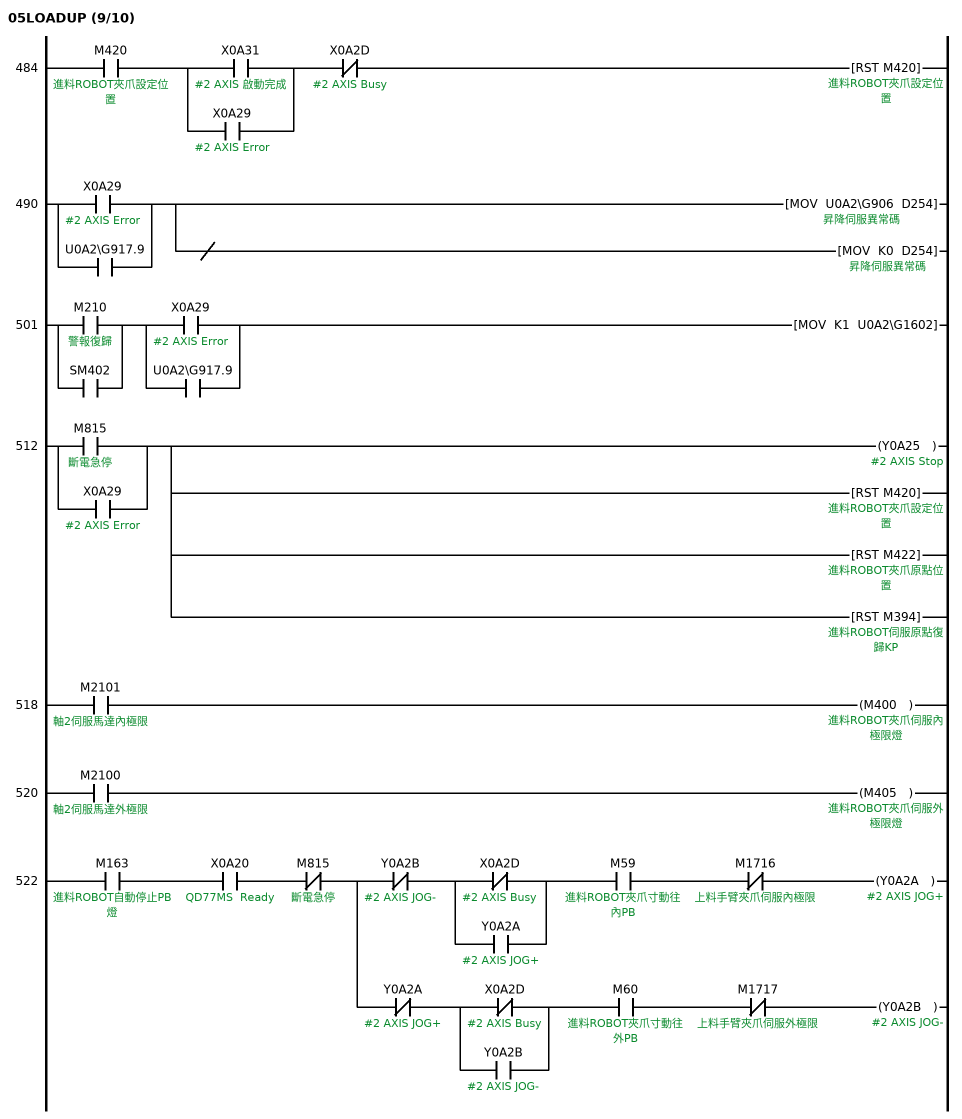
[picture p24: ladder of 05LOADUP, rungs at steps 484 to 522]
484   LD      M420  ; 進料ROBOT夾爪設定位置
      LD      X0A31  ; #2 AXIS 啟動完成
      OR      X0A29  ; #2 AXIS Error
      ANB
      ANI     X0A2D  ; #2 AXIS Busy
      RST     M420  ; 進料ROBOT夾爪設定位置
490   LD      X0A29  ; #2 AXIS Error
      OR      U0A2\G917.9
      MOV     U0A2\G906 D254  ; 昇降伺服異常碼
      INV
      MOV     K0 D254
501   LD      M210  ; 警報復歸
      OR      SM402
      LD      X0A29  ; #2 AXIS Error
      OR      U0A2\G917.9
      ANB
      MOV     K1 U0A2\G1602
512   LD      M815  ; 斷電急停
      OR      X0A29  ; #2 AXIS Error
      OUT     Y0A25  ; #2 AXIS Stop
      RST     M420  ; 進料ROBOT夾爪設定位置
      RST     M422  ; 進料ROBOT夾爪原點位置
      RST     M394  ; 進料ROBOT伺服原點復歸KP
518   LD      M2101  ; 軸2伺服馬達內極限
      OUT     M400  ; 進料ROBOT夾爪伺服內極限燈
520   LD      M2100  ; 軸2伺服馬達外極限
      OUT     M405  ; 進料ROBOT夾爪伺服外極限燈
522   LD      M163  ; 進料ROBOT自動停止PB燈
      AND     X0A20  ; QD77MS  Ready
      ANI     M815  ; 斷電急停
      MPS
      ANI     Y0A2B  ; #2 AXIS JOG-
      LDI     X0A2D  ; #2 AXIS Busy
      OR      Y0A2A  ; #2 AXIS JOG+
      ANB
      AND     M59  ; 進料ROBOT夾爪寸動往內PB
      ANI     M1716  ; 上料手臂夾爪伺服內極限
      OUT     Y0A2A  ; #2 AXIS JOG+
      MPP
      ANI     Y0A2A  ; #2 AXIS JOG+
      LDI     X0A2D  ; #2 AXIS Busy
      OR      Y0A2B  ; #2 AXIS JOG-
      ANB
      AND     M60  ; 進料ROBOT夾爪寸動往外PB
      ANI     M1717  ; 上料手臂夾爪伺服外極限
      OUT     Y0A2B  ; #2 AXIS JOG-
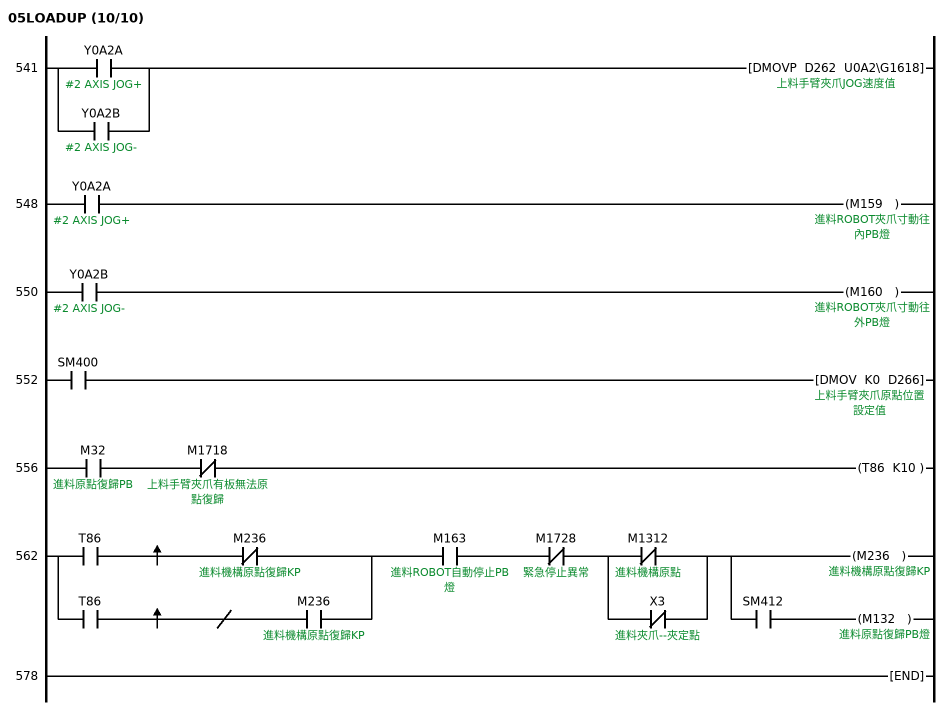
541   LD      Y0A2A  ; #2 AXIS JOG+
      OR      Y0A2B  ; #2 AXIS JOG-
      DMOVP   D262 U0A2\G1618  ; 上料手臂夾爪JOG速度值
548   LD      Y0A2A  ; #2 AXIS JOG+
      OUT     M159  ; 進料ROBOT夾爪寸動往內PB燈
550   LD      Y0A2B  ; #2 AXIS JOG-
      OUT     M160  ; 進料ROBOT夾爪寸動往外PB燈
552   LD      SM400
      DMOV    K0 D266
556   LD      M32  ; 進料原點復歸PB
      ANI     M1718  ; 上料手臂夾爪有板無法原點復歸
      OUT     T86 K10
562   LD      T86
      MEP
      ANI     M236  ; 進料機構原點復歸KP
      LD      T86
      MEP
      INV
      AND     M236  ; 進料機構原點復歸KP
      ORB
      AND     M163  ; 進料ROBOT自動停止PB燈
      ANI     M1728  ; 緊急停止異常
      LDI     M1312  ; 進料機構原點
      ORI     X3  ; 進料夾爪--夾定點
      ANB
      OUT     M236  ; 進料機構原點復歸KP
      AND     SM412
      OUT     M132  ; 進料原點復歸PB燈
578   END
END_PROGRAM

PROGRAM 06UNLOAD
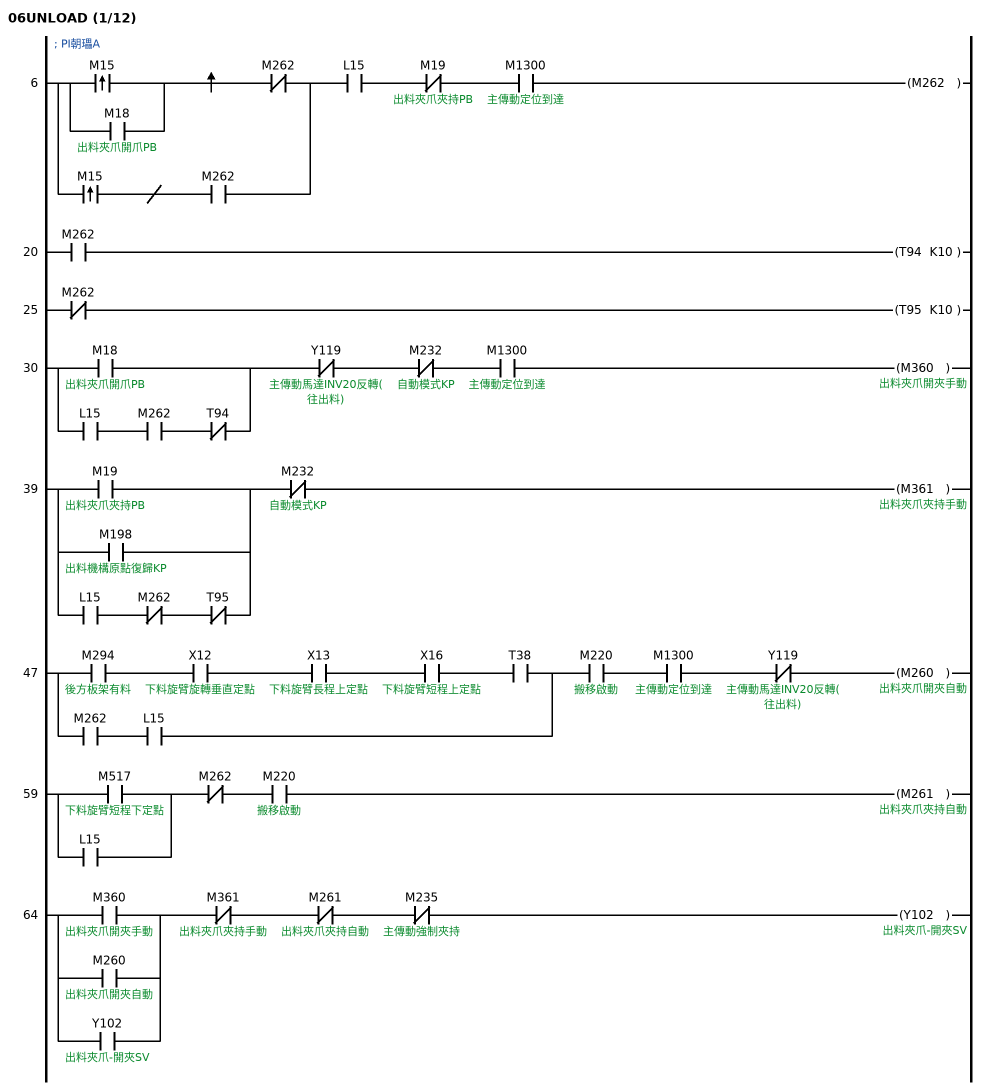
; PI朝瓃Α
6     LDP     M15
      OR      M18  ; 出料夾爪開爪PB
      MEP
      ANI     M262
      LDP     M15
      INV
      AND     M262
      ORB
      AND     L15
      ANI     M19  ; 出料夾爪夾持PB
      AND     M1300  ; 主傳動定位到達
      OUT     M262
20    LD      M262
      OUT     T94 K10
25    LDI     M262
      OUT     T95 K10
30    LD      M18  ; 出料夾爪開爪PB
      LD      L15
      AND     M262
      ANI     T94
      ORB
      ANI     Y119  ; 主傳動馬達INV20反轉(往出料)
      ANI     M232  ; 自動模式KP
      AND     M1300  ; 主傳動定位到達
      OUT     M360  ; 出料夾爪開夾手動
39    LD      M19  ; 出料夾爪夾持PB
      OR      M198  ; 出料機構原點復歸KP
      LD      L15
      ANI     M262
      ANI     T95
      ORB
      ANI     M232  ; 自動模式KP
      OUT     M361  ; 出料夾爪夾持手動
47    LD      M294  ; 後方板架有料
      AND     X12  ; 下料旋臂旋轉垂直定點
      AND     X13  ; 下料旋臂長程上定點
      AND     X16  ; 下料旋臂短程上定點
      AND     T38
      LD      M262
      AND     L15
      ORB
      AND     M220  ; 搬移啟動
      AND     M1300  ; 主傳動定位到達
      ANI     Y119  ; 主傳動馬達INV20反轉(往出料)
      OUT     M260  ; 出料夾爪開夾自動
59    LD      M517  ; 下料旋臂短程下定點
      OR      L15
      ANI     M262
      AND     M220  ; 搬移啟動
      OUT     M261  ; 出料夾爪夾持自動
64    LD      M360  ; 出料夾爪開夾手動
      OR      M260  ; 出料夾爪開夾自動
      OR      Y102  ; 出料夾爪-開夾SV
      ANI     M361  ; 出料夾爪夾持手動
      ANI     M261  ; 出料夾爪夾持自動
      ANI     M235  ; 主傳動強制夾持
      OUT     Y102  ; 出料夾爪-開夾SV
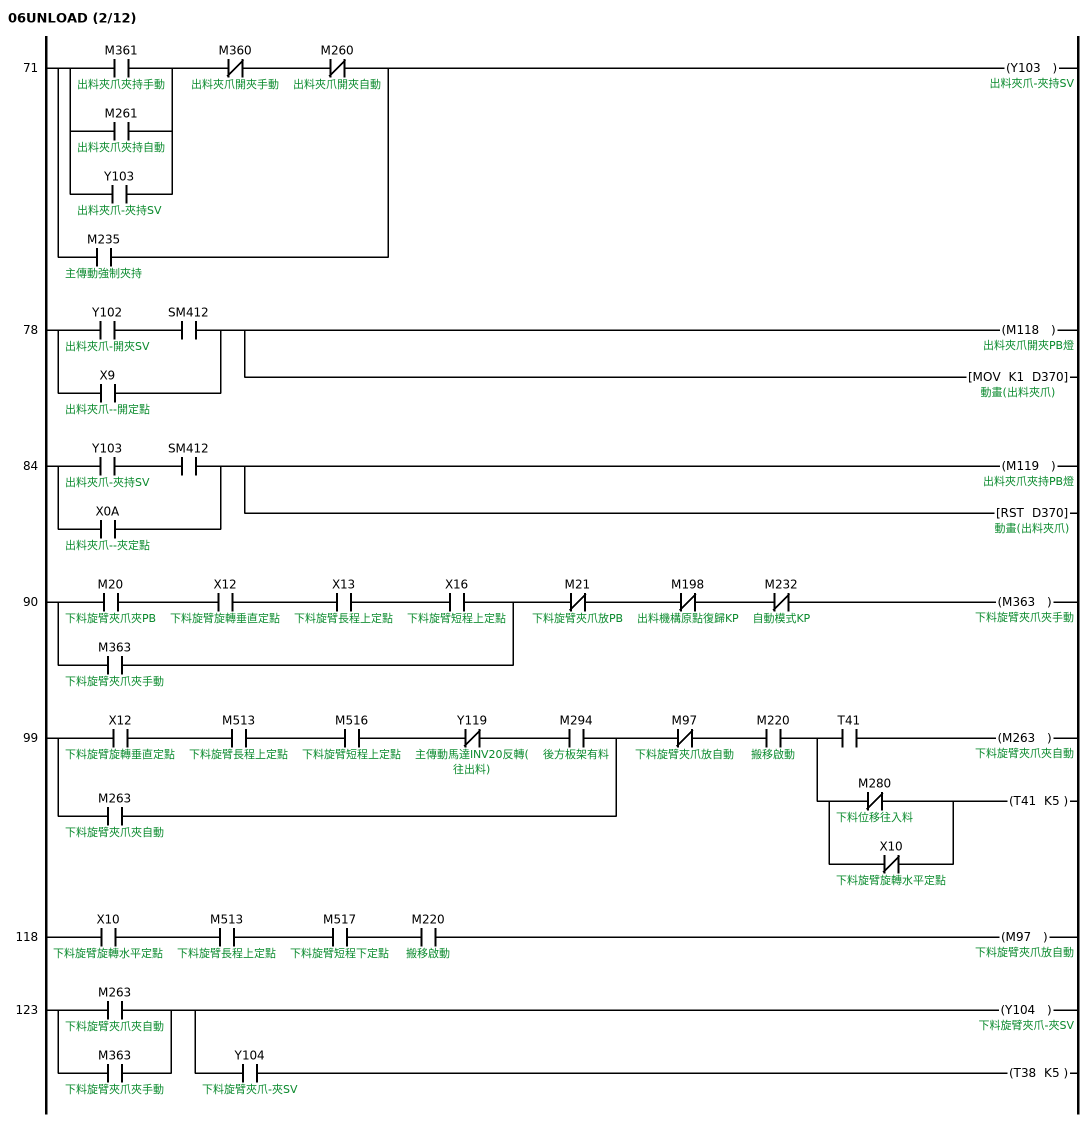
71    LD      M361  ; 出料夾爪夾持手動
      OR      M261  ; 出料夾爪夾持自動
      OR      Y103  ; 出料夾爪-夾持SV
      ANI     M360  ; 出料夾爪開夾手動
      ANI     M260  ; 出料夾爪開夾自動
      OR      M235  ; 主傳動強制夾持
      OUT     Y103  ; 出料夾爪-夾持SV
78    LD      Y102  ; 出料夾爪-開夾SV
      AND     SM412
      OR      X9  ; 出料夾爪--開定點
      OUT     M118  ; 出料夾爪開夾PB燈
      MOV     K1 D370  ; 動畫(出料夾爪)
84    LD      Y103  ; 出料夾爪-夾持SV
      AND     SM412
      OR      X0A  ; 出料夾爪--夾定點
      OUT     M119  ; 出料夾爪夾持PB燈
      RST     D370  ; 動畫(出料夾爪)
90    LD      M20  ; 下料旋臂夾爪夾PB
      AND     X12  ; 下料旋臂旋轉垂直定點
      AND     X13  ; 下料旋臂長程上定點
      AND     X16  ; 下料旋臂短程上定點
      OR      M363  ; 下料旋臂夾爪夾手動
      ANI     M21  ; 下料旋臂夾爪放PB
      ANI     M198  ; 出料機構原點復歸KP
      ANI     M232  ; 自動模式KP
      OUT     M363  ; 下料旋臂夾爪夾手動
99    LD      X12  ; 下料旋臂旋轉垂直定點
      AND     M513  ; 下料旋臂長程上定點
      AND     M516  ; 下料旋臂短程上定點
      ANI     Y119  ; 主傳動馬達INV20反轉(往出料)
      AND     M294  ; 後方板架有料
      OR      M263  ; 下料旋臂夾爪夾自動
      ANI     M97  ; 下料旋臂夾爪放自動
      AND     M220  ; 搬移啟動
      MPS
      AND     T41
      OUT     M263  ; 下料旋臂夾爪夾自動
      MPP
      LDI     M280  ; 下料位移往入料
      ORI     X10  ; 下料旋臂旋轉水平定點
      ANB
      OUT     T41 K5
118   LD      X10  ; 下料旋臂旋轉水平定點
      AND     M513  ; 下料旋臂長程上定點
      AND     M517  ; 下料旋臂短程下定點
      AND     M220  ; 搬移啟動
      OUT     M97  ; 下料旋臂夾爪放自動
123   LD      M263  ; 下料旋臂夾爪夾自動
      OR      M363  ; 下料旋臂夾爪夾手動
      OUT     Y104  ; 下料旋臂夾爪-夾SV
      AND     Y104  ; 下料旋臂夾爪-夾SV
      OUT     T38 K5
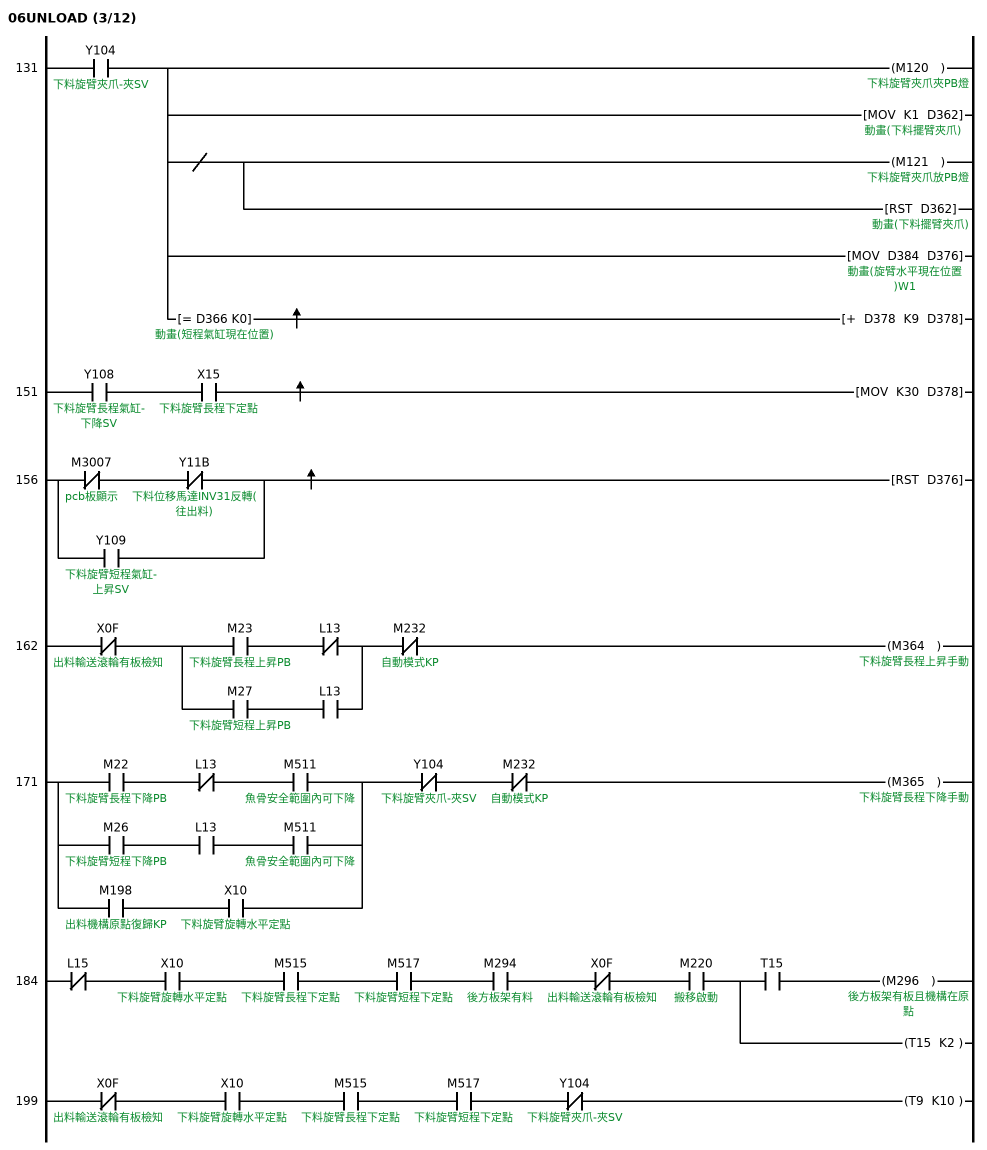
131   LD      Y104  ; 下料旋臂夾爪-夾SV
      OUT     M120  ; 下料旋臂夾爪夾PB燈
      MOV     K1 D362  ; 動畫(下料擺臂夾爪)
      MPS
      INV
      OUT     M121  ; 下料旋臂夾爪放PB燈
      RST     D362  ; 動畫(下料擺臂夾爪)
      MPP
      MOV     D384 D376  ; 動畫(旋臂水平現在位置)W1
      AND=    D366 K0  ; 動畫(短程氣缸現在位置)
      MEP
      +       D378 K9 D378
151   LD      Y108  ; 下料旋臂長程氣缸-下降SV
      AND     X15  ; 下料旋臂長程下定點
      MEP
      MOV     K30 D378
156   LDI     M3007  ; pcb板顯示
      ANI     Y11B  ; 下料位移馬達INV31反轉(往出料)
      OR      Y109  ; 下料旋臂短程氣缸-上昇SV
      MEP
      RST     D376
162   LDI     X0F  ; 出料輸送滾輪有板檢知
      LD      M23  ; 下料旋臂長程上昇PB
      ANI     L13
      LD      M27  ; 下料旋臂短程上昇PB
      AND     L13
      ORB
      ANB
      ANI     M232  ; 自動模式KP
      OUT     M364  ; 下料旋臂長程上昇手動
171   LD      M22  ; 下料旋臂長程下降PB
      ANI     L13
      AND     M511  ; 魚骨安全範圍內可下降
      LD      M26  ; 下料旋臂短程下降PB
      AND     L13
      AND     M511  ; 魚骨安全範圍內可下降
      ORB
      LD      M198  ; 出料機構原點復歸KP
      AND     X10  ; 下料旋臂旋轉水平定點
      ORB
      ANI     Y104  ; 下料旋臂夾爪-夾SV
      ANI     M232  ; 自動模式KP
      OUT     M365  ; 下料旋臂長程下降手動
184   LDI     L15
      AND     X10  ; 下料旋臂旋轉水平定點
      AND     M515  ; 下料旋臂長程下定點
      AND     M517  ; 下料旋臂短程下定點
      AND     M294  ; 後方板架有料
      ANI     X0F  ; 出料輸送滾輪有板檢知
      AND     M220  ; 搬移啟動
      MPS
      AND     T15
      OUT     M296  ; 後方板架有板且機構在原點
      MPP
      OUT     T15 K2
199   LDI     X0F  ; 出料輸送滾輪有板檢知
      AND     X10  ; 下料旋臂旋轉水平定點
      AND     M515  ; 下料旋臂長程下定點
      AND     M517  ; 下料旋臂短程下定點
      ANI     Y104  ; 下料旋臂夾爪-夾SV
      OUT     T9 K10
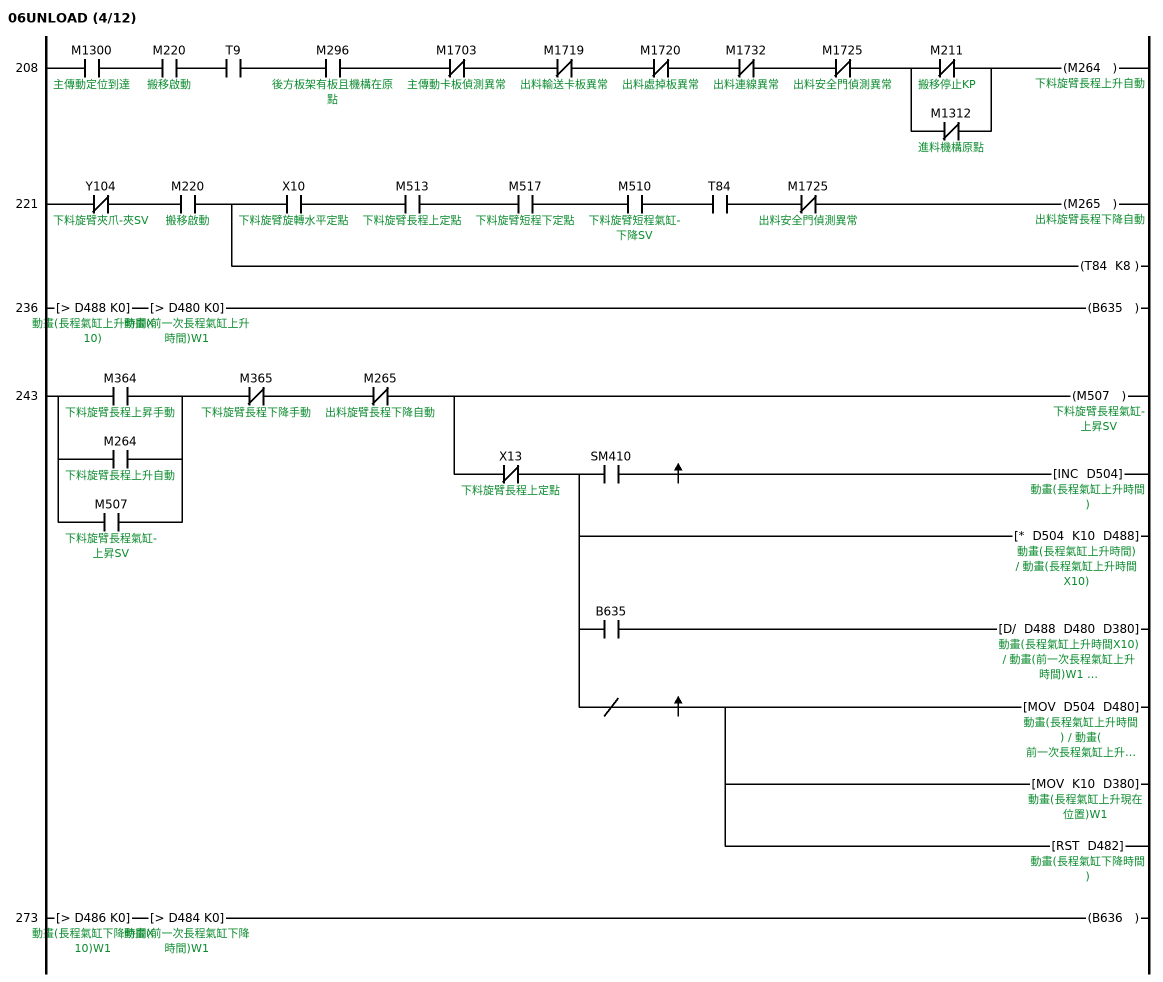
208   LD      M1300  ; 主傳動定位到達
      AND     M220  ; 搬移啟動
      AND     T9
      AND     M296  ; 後方板架有板且機構在原點
      ANI     M1703  ; 主傳動卡板偵測異常
      ANI     M1719  ; 出料輸送卡板異常
      ANI     M1720  ; 出料處掉板異常
      ANI     M1732  ; 出料連線異常
      ANI     M1725  ; 出料安全門偵測異常
      LDI     M211  ; 搬移停止KP
      ORI     M1312  ; 進料機構原點
      ANB
      OUT     M264  ; 下料旋臂長程上升自動
221   LDI     Y104  ; 下料旋臂夾爪-夾SV
      AND     M220  ; 搬移啟動
      MPS
      AND     X10  ; 下料旋臂旋轉水平定點
      AND     M513  ; 下料旋臂長程上定點
      AND     M517  ; 下料旋臂短程下定點
      AND     M510  ; 下料旋臂短程氣缸-下降SV
      AND     T84
      ANI     M1725  ; 出料安全門偵測異常
      OUT     M265  ; 出料旋臂長程下降自動
      MPP
      OUT     T84 K8
236   LD>     D488 K0  ; 動畫(長程氣缸上升時間X10)
      AND>    D480 K0  ; 動畫(前一次長程氣缸上升時間)W1
      OUT     B635
243   LD      M364  ; 下料旋臂長程上昇手動
      OR      M264  ; 下料旋臂長程上升自動
      OR      M507  ; 下料旋臂長程氣缸-上昇SV
      ANI     M365  ; 下料旋臂長程下降手動
      ANI     M265  ; 出料旋臂長程下降自動
      OUT     M507  ; 下料旋臂長程氣缸-上昇SV
      ANI     X13  ; 下料旋臂長程上定點
      MPS
      AND     SM410
      MEP
      INC     D504  ; 動畫(長程氣缸上升時間)
      MPP
      *       D504 K10 D488
      MPS
      AND     B635
      D/      D488 D480 D380  ; 動畫(長程氣缸上升現在位置)W1
      MPP
      INV
      MEP
      MOV     D504 D480
      MOV     K10 D380
      RST     D482  ; 動畫(長程氣缸下降時間)
273   LD>     D486 K0  ; 動畫(長程氣缸下降時間X10)W1
      AND>    D484 K0  ; 動畫(前一次長程氣缸下降時間)W1
      OUT     B636
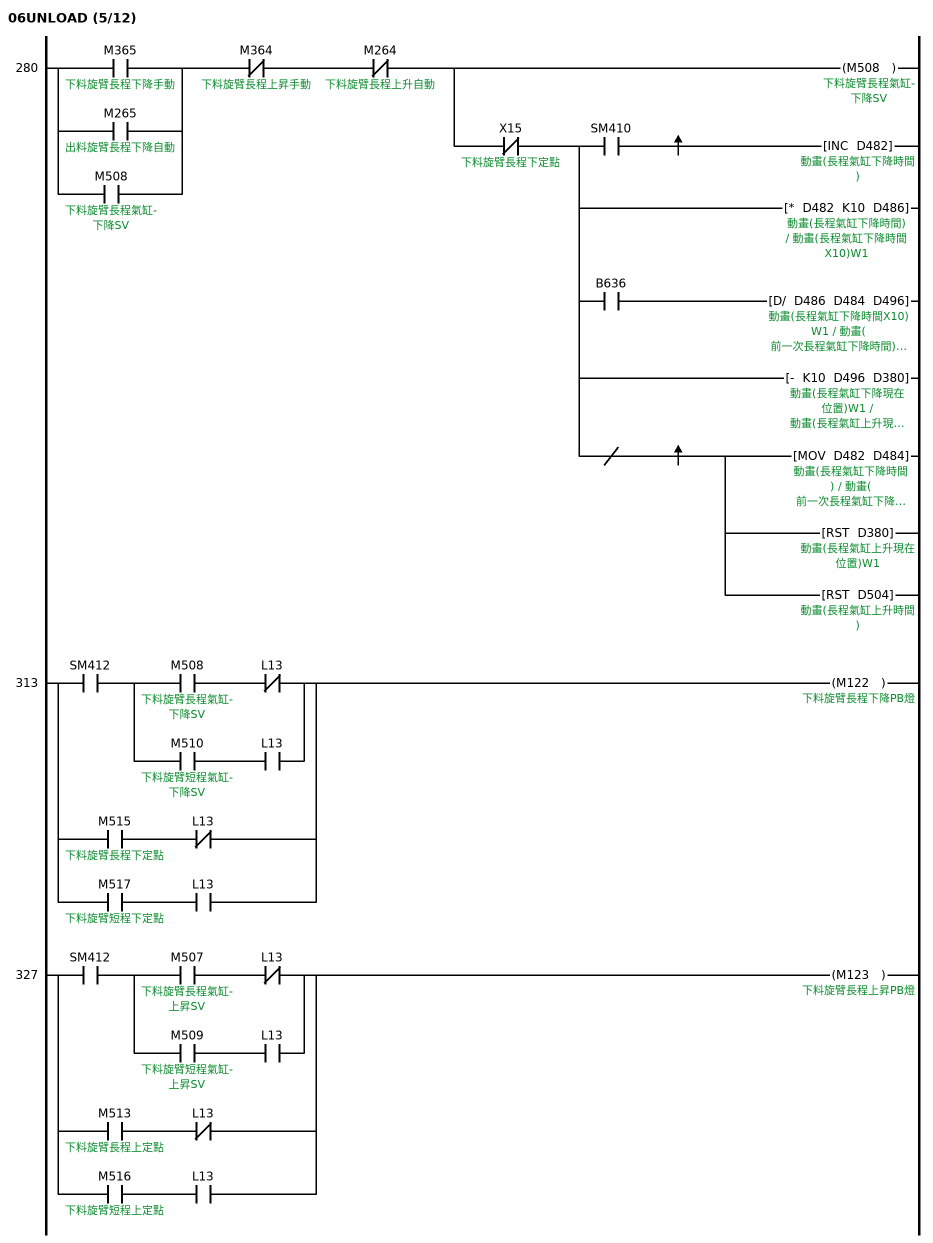
280   LD      M365  ; 下料旋臂長程下降手動
      OR      M265  ; 出料旋臂長程下降自動
      OR      M508  ; 下料旋臂長程氣缸-下降SV
      ANI     M364  ; 下料旋臂長程上昇手動
      ANI     M264  ; 下料旋臂長程上升自動
      OUT     M508  ; 下料旋臂長程氣缸-下降SV
      ANI     X15  ; 下料旋臂長程下定點
      MPS
      AND     SM410
      MEP
      INC     D482
      MPP
      *       D482 K10 D486
      MPS
      AND     B636
      D/      D486 D484 D496  ; 動畫(長程氣缸下降現在位置)W1
      MPP
      -       K10 D496 D380
      INV
      MEP
      MOV     D482 D484
      RST     D380  ; 動畫(長程氣缸上升現在位置)W1
      RST     D504  ; 動畫(長程氣缸上升時間)
313   LD      SM412
      LD      M508  ; 下料旋臂長程氣缸-下降SV
      ANI     L13
      LD      M510  ; 下料旋臂短程氣缸-下降SV
      AND     L13
      ORB
      ANB
      LD      M515  ; 下料旋臂長程下定點
      ANI     L13
      ORB
      LD      M517  ; 下料旋臂短程下定點
      AND     L13
      ORB
      OUT     M122  ; 下料旋臂長程下降PB燈
327   LD      SM412
      LD      M507  ; 下料旋臂長程氣缸-上昇SV
      ANI     L13
      LD      M509  ; 下料旋臂短程氣缸-上昇SV
      AND     L13
      ORB
      ANB
      LD      M513  ; 下料旋臂長程上定點
      ANI     L13
      ORB
      LD      M516  ; 下料旋臂短程上定點
      AND     L13
      ORB
      OUT     M123  ; 下料旋臂長程上昇PB燈
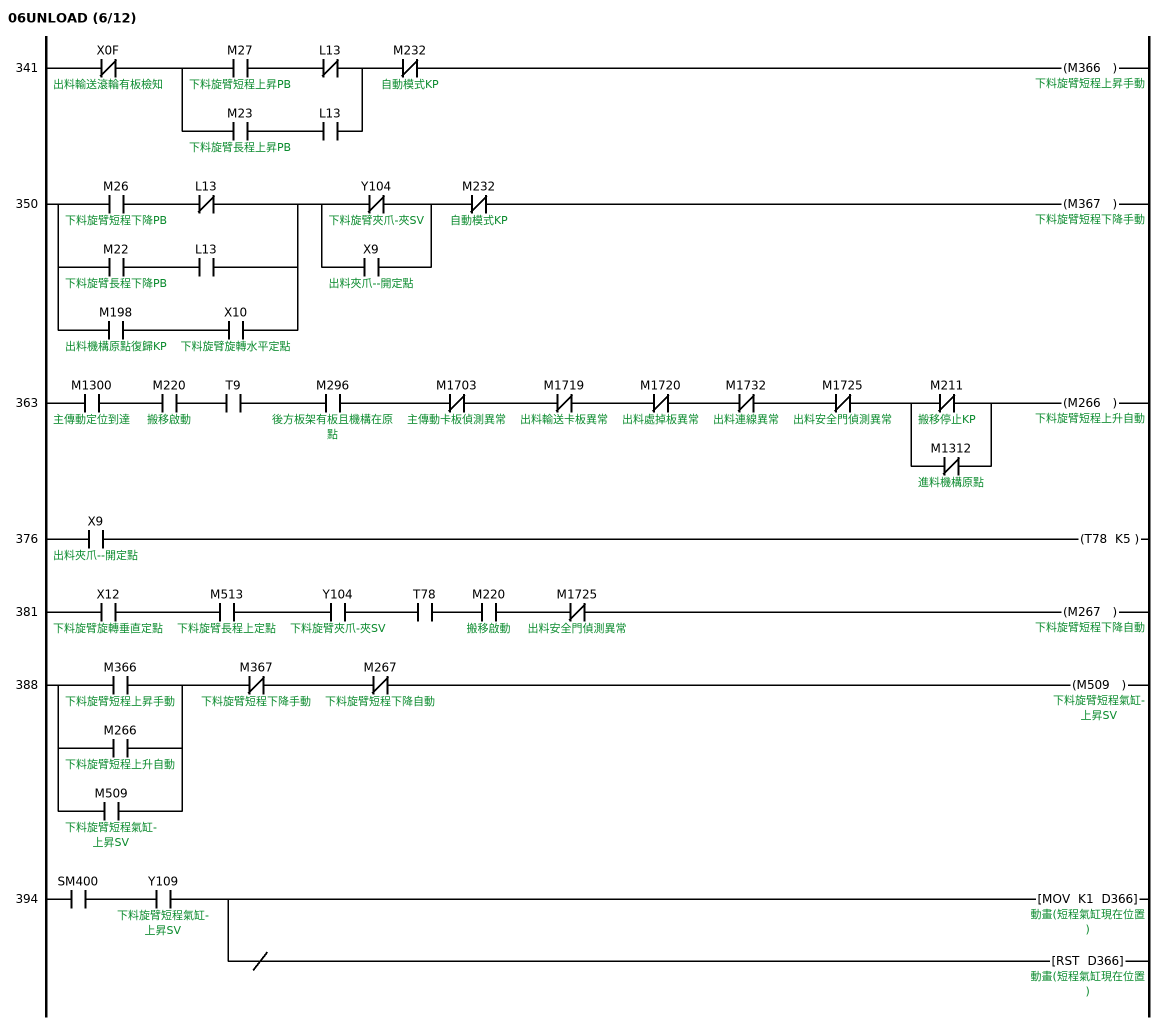
341   LDI     X0F  ; 出料輸送滾輪有板檢知
      LD      M27  ; 下料旋臂短程上昇PB
      ANI     L13
      LD      M23  ; 下料旋臂長程上昇PB
      AND     L13
      ORB
      ANB
      ANI     M232  ; 自動模式KP
      OUT     M366  ; 下料旋臂短程上昇手動
350   LD      M26  ; 下料旋臂短程下降PB
      ANI     L13
      LD      M22  ; 下料旋臂長程下降PB
      AND     L13
      ORB
      LD      M198  ; 出料機構原點復歸KP
      AND     X10  ; 下料旋臂旋轉水平定點
      ORB
      LDI     Y104  ; 下料旋臂夾爪-夾SV
      OR      X9  ; 出料夾爪--開定點
      ANB
      ANI     M232  ; 自動模式KP
      OUT     M367  ; 下料旋臂短程下降手動
363   LD      M1300  ; 主傳動定位到達
      AND     M220  ; 搬移啟動
      AND     T9
      AND     M296  ; 後方板架有板且機構在原點
      ANI     M1703  ; 主傳動卡板偵測異常
      ANI     M1719  ; 出料輸送卡板異常
      ANI     M1720  ; 出料處掉板異常
      ANI     M1732  ; 出料連線異常
      ANI     M1725  ; 出料安全門偵測異常
      LDI     M211  ; 搬移停止KP
      ORI     M1312  ; 進料機構原點
      ANB
      OUT     M266  ; 下料旋臂短程上升自動
376   LD      X9  ; 出料夾爪--開定點
      OUT     T78 K5
381   LD      X12  ; 下料旋臂旋轉垂直定點
      AND     M513  ; 下料旋臂長程上定點
      AND     Y104  ; 下料旋臂夾爪-夾SV
      AND     T78
      AND     M220  ; 搬移啟動
      ANI     M1725  ; 出料安全門偵測異常
      OUT     M267  ; 下料旋臂短程下降自動
388   LD      M366  ; 下料旋臂短程上昇手動
      OR      M266  ; 下料旋臂短程上升自動
      OR      M509  ; 下料旋臂短程氣缸-上昇SV
      ANI     M367  ; 下料旋臂短程下降手動
      ANI     M267  ; 下料旋臂短程下降自動
      OUT     M509  ; 下料旋臂短程氣缸-上昇SV
394   LD      SM400
      AND     Y109  ; 下料旋臂短程氣缸-上昇SV
      MOV     K1 D366
      INV
      RST     D366  ; 動畫(短程氣缸現在位置)
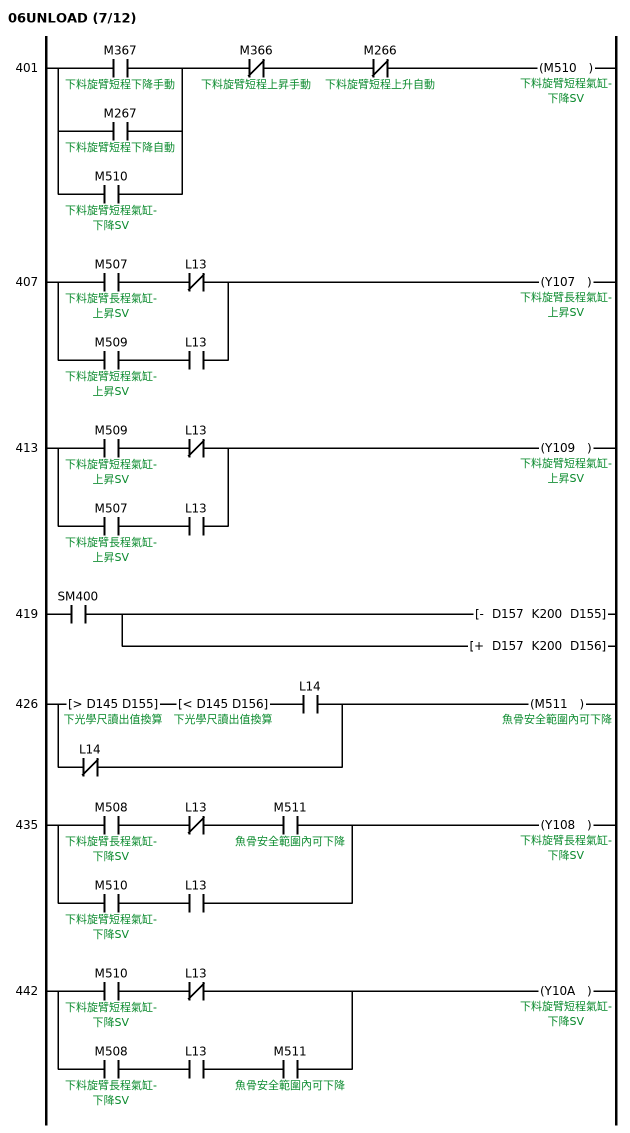
401   LD      M367  ; 下料旋臂短程下降手動
      OR      M267  ; 下料旋臂短程下降自動
      OR      M510  ; 下料旋臂短程氣缸-下降SV
      ANI     M366  ; 下料旋臂短程上昇手動
      ANI     M266  ; 下料旋臂短程上升自動
      OUT     M510  ; 下料旋臂短程氣缸-下降SV
407   LD      M507  ; 下料旋臂長程氣缸-上昇SV
      ANI     L13
      LD      M509  ; 下料旋臂短程氣缸-上昇SV
      AND     L13
      ORB
      OUT     Y107  ; 下料旋臂長程氣缸-上昇SV
413   LD      M509  ; 下料旋臂短程氣缸-上昇SV
      ANI     L13
      LD      M507  ; 下料旋臂長程氣缸-上昇SV
      AND     L13
      ORB
      OUT     Y109  ; 下料旋臂短程氣缸-上昇SV
419   LD      SM400
      -       D157 K200 D155
      +       D157 K200 D156
426   LD>     D145 D155  ; 下光學尺讀出值換算
      AND<    D145 D156  ; 下光學尺讀出值換算
      AND     L14
      ORI     L14
      OUT     M511  ; 魚骨安全範圍內可下降
435   LD      M508  ; 下料旋臂長程氣缸-下降SV
      ANI     L13
      AND     M511  ; 魚骨安全範圍內可下降
      LD      M510  ; 下料旋臂短程氣缸-下降SV
      AND     L13
      ORB
      OUT     Y108  ; 下料旋臂長程氣缸-下降SV
442   LD      M510  ; 下料旋臂短程氣缸-下降SV
      ANI     L13
      LD      M508  ; 下料旋臂長程氣缸-下降SV
      AND     L13
      AND     M511  ; 魚骨安全範圍內可下降
      ORB
      OUT     Y10A  ; 下料旋臂短程氣缸-下降SV
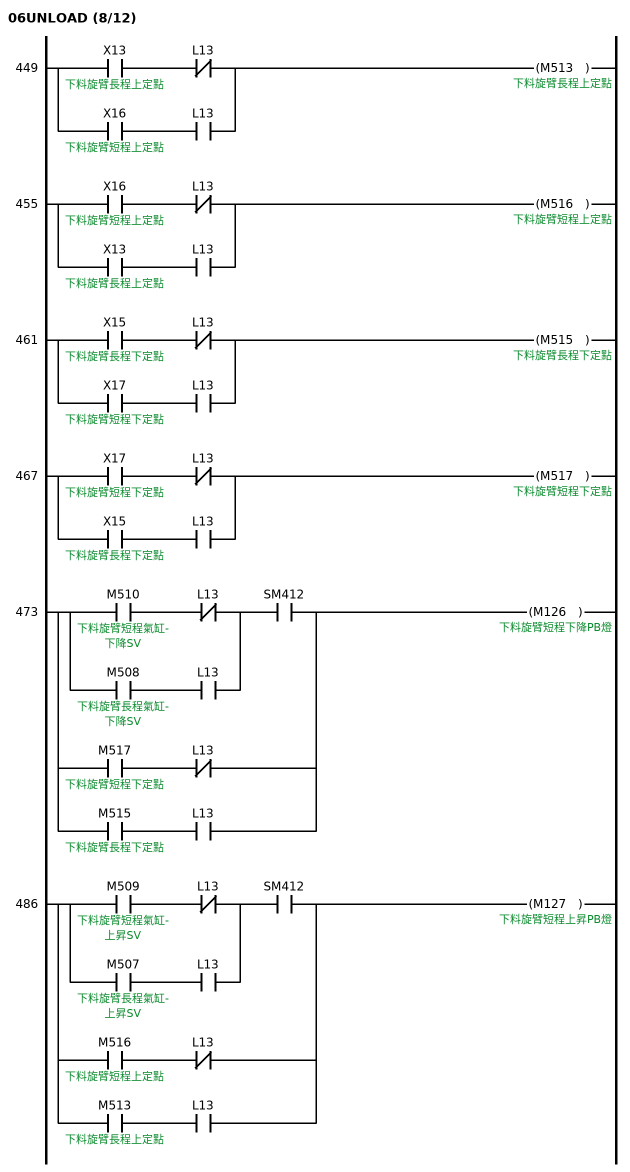
449   LD      X13  ; 下料旋臂長程上定點
      ANI     L13
      LD      X16  ; 下料旋臂短程上定點
      AND     L13
      ORB
      OUT     M513  ; 下料旋臂長程上定點
455   LD      X16  ; 下料旋臂短程上定點
      ANI     L13
      LD      X13  ; 下料旋臂長程上定點
      AND     L13
      ORB
      OUT     M516  ; 下料旋臂短程上定點
461   LD      X15  ; 下料旋臂長程下定點
      ANI     L13
      LD      X17  ; 下料旋臂短程下定點
      AND     L13
      ORB
      OUT     M515  ; 下料旋臂長程下定點
467   LD      X17  ; 下料旋臂短程下定點
      ANI     L13
      LD      X15  ; 下料旋臂長程下定點
      AND     L13
      ORB
      OUT     M517  ; 下料旋臂短程下定點
473   LD      M510  ; 下料旋臂短程氣缸-下降SV
      ANI     L13
      LD      M508  ; 下料旋臂長程氣缸-下降SV
      AND     L13
      ORB
      AND     SM412
      LD      M517  ; 下料旋臂短程下定點
      ANI     L13
      ORB
      LD      M515  ; 下料旋臂長程下定點
      AND     L13
      ORB
      OUT     M126  ; 下料旋臂短程下降PB燈
486   LD      M509  ; 下料旋臂短程氣缸-上昇SV
      ANI     L13
      LD      M507  ; 下料旋臂長程氣缸-上昇SV
      AND     L13
      ORB
      AND     SM412
      LD      M516  ; 下料旋臂短程上定點
      ANI     L13
      ORB
      LD      M513  ; 下料旋臂長程上定點
      AND     L13
      ORB
      OUT     M127  ; 下料旋臂短程上昇PB燈
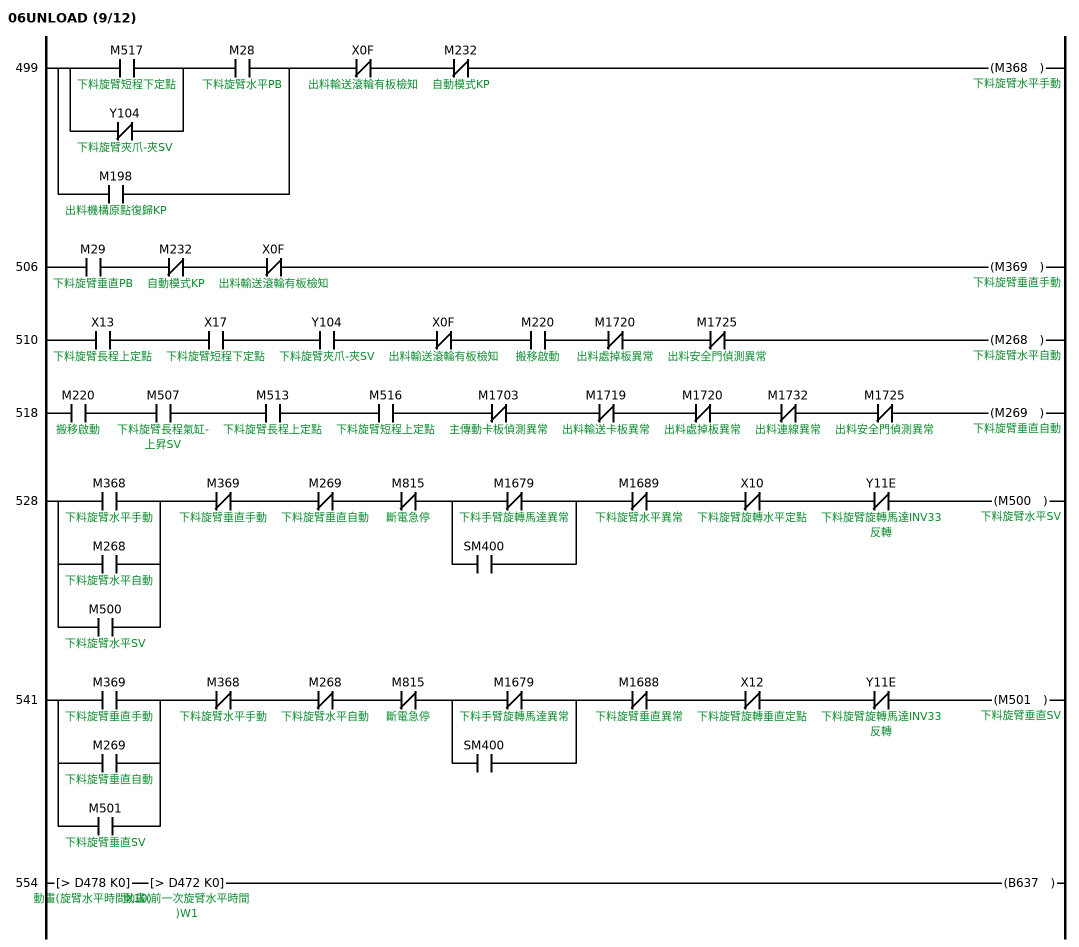
499   LD      M517  ; 下料旋臂短程下定點
      ORI     Y104  ; 下料旋臂夾爪-夾SV
      AND     M28  ; 下料旋臂水平PB
      OR      M198  ; 出料機構原點復歸KP
      ANI     X0F  ; 出料輸送滾輪有板檢知
      ANI     M232  ; 自動模式KP
      OUT     M368  ; 下料旋臂水平手動
506   LD      M29  ; 下料旋臂垂直PB
      ANI     M232  ; 自動模式KP
      ANI     X0F  ; 出料輸送滾輪有板檢知
      OUT     M369  ; 下料旋臂垂直手動
510   LD      X13  ; 下料旋臂長程上定點
      AND     X17  ; 下料旋臂短程下定點
      AND     Y104  ; 下料旋臂夾爪-夾SV
      ANI     X0F  ; 出料輸送滾輪有板檢知
      AND     M220  ; 搬移啟動
      ANI     M1720  ; 出料處掉板異常
      ANI     M1725  ; 出料安全門偵測異常
      OUT     M268  ; 下料旋臂水平自動
518   LD      M220  ; 搬移啟動
      AND     M507  ; 下料旋臂長程氣缸-上昇SV
      AND     M513  ; 下料旋臂長程上定點
      AND     M516  ; 下料旋臂短程上定點
      ANI     M1703  ; 主傳動卡板偵測異常
      ANI     M1719  ; 出料輸送卡板異常
      ANI     M1720  ; 出料處掉板異常
      ANI     M1732  ; 出料連線異常
      ANI     M1725  ; 出料安全門偵測異常
      OUT     M269  ; 下料旋臂垂直自動
528   LD      M368  ; 下料旋臂水平手動
      OR      M268  ; 下料旋臂水平自動
      OR      M500  ; 下料旋臂水平SV
      ANI     M369  ; 下料旋臂垂直手動
      ANI     M269  ; 下料旋臂垂直自動
      ANI     M815  ; 斷電急停
      LDI     M1679  ; 下料手臂旋轉馬達異常
      OR      SM400
      ANB
      ANI     M1689  ; 下料旋臂水平異常
      ANI     X10  ; 下料旋臂旋轉水平定點
      ANI     Y11E  ; 下料旋臂旋轉馬達INV33反轉
      OUT     M500  ; 下料旋臂水平SV
541   LD      M369  ; 下料旋臂垂直手動
      OR      M269  ; 下料旋臂垂直自動
      OR      M501  ; 下料旋臂垂直SV
      ANI     M368  ; 下料旋臂水平手動
      ANI     M268  ; 下料旋臂水平自動
      ANI     M815  ; 斷電急停
      LDI     M1679  ; 下料手臂旋轉馬達異常
      OR      SM400
      ANB
      ANI     M1688  ; 下料旋臂垂直異常
      ANI     X12  ; 下料旋臂旋轉垂直定點
      ANI     Y11E  ; 下料旋臂旋轉馬達INV33反轉
      OUT     M501  ; 下料旋臂垂直SV
554   LD>     D478 K0  ; 動畫(旋臂水平時間X10)
      AND>    D472 K0  ; 動畫(前一次旋臂水平時間)W1
      OUT     B637
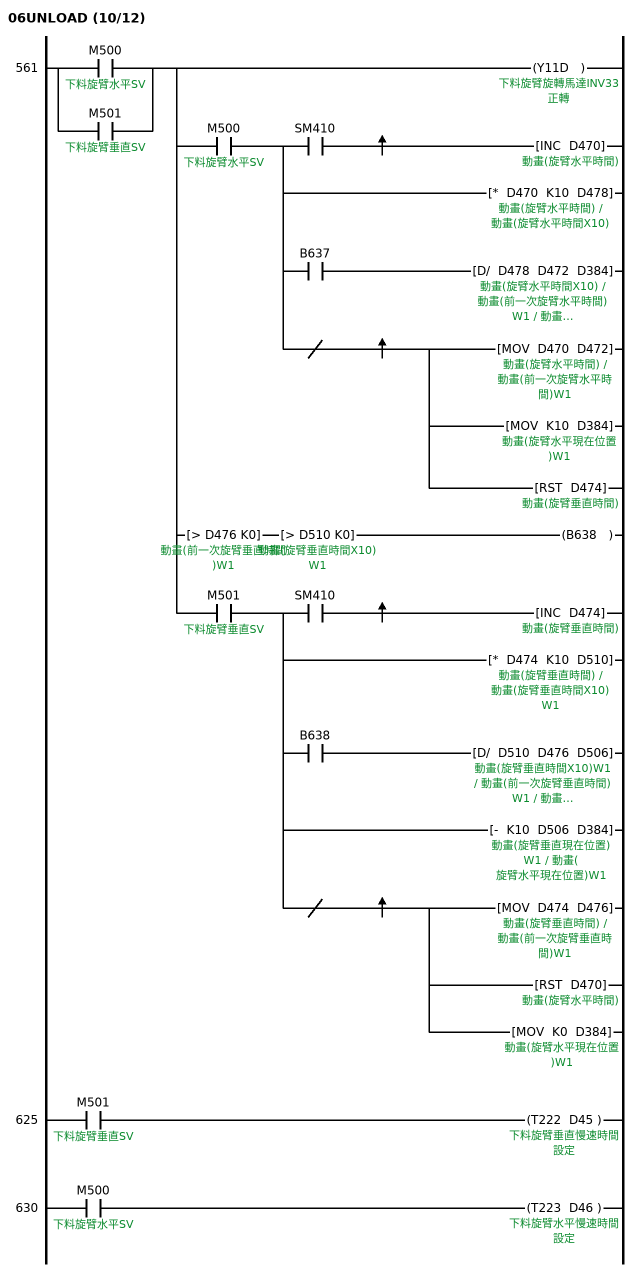
561   LD      M500  ; 下料旋臂水平SV
      OR      M501  ; 下料旋臂垂直SV
      OUT     Y11D  ; 下料旋臂旋轉馬達INV33正轉
      MPS
      AND     M500  ; 下料旋臂水平SV
      MPS
      AND     SM410
      MEP
      INC     D470  ; 動畫(旋臂水平時間)
      MPP
      *       D470 K10 D478
      MPS
      AND     B637
      D/      D478 D472 D384
      MPP
      INV
      MEP
      MOV     D470 D472
      MOV     K10 D384
      RST     D474  ; 動畫(旋臂垂直時間)
      MRD
      AND>    D476 K0  ; 動畫(前一次旋臂垂直時間)W1
      AND>    D510 K0  ; 動畫(旋臂垂直時間X10)W1
      OUT     B638
      MPP
      AND     M501  ; 下料旋臂垂直SV
      MPS
      AND     SM410
      MEP
      INC     D474
      MPP
      *       D474 K10 D510
      MPS
      AND     B638
      D/      D510 D476 D506  ; 動畫(旋臂垂直現在位置)W1
      MPP
      -       K10 D506 D384
      INV
      MEP
      MOV     D474 D476
      RST     D470  ; 動畫(旋臂水平時間)
      MOV     K0 D384
625   LD      M501  ; 下料旋臂垂直SV
      OUT     T222 D45  ; 下料旋臂垂直慢速時間設定
630   LD      M500  ; 下料旋臂水平SV
      OUT     T223 D46  ; 下料旋臂水平慢速時間設定
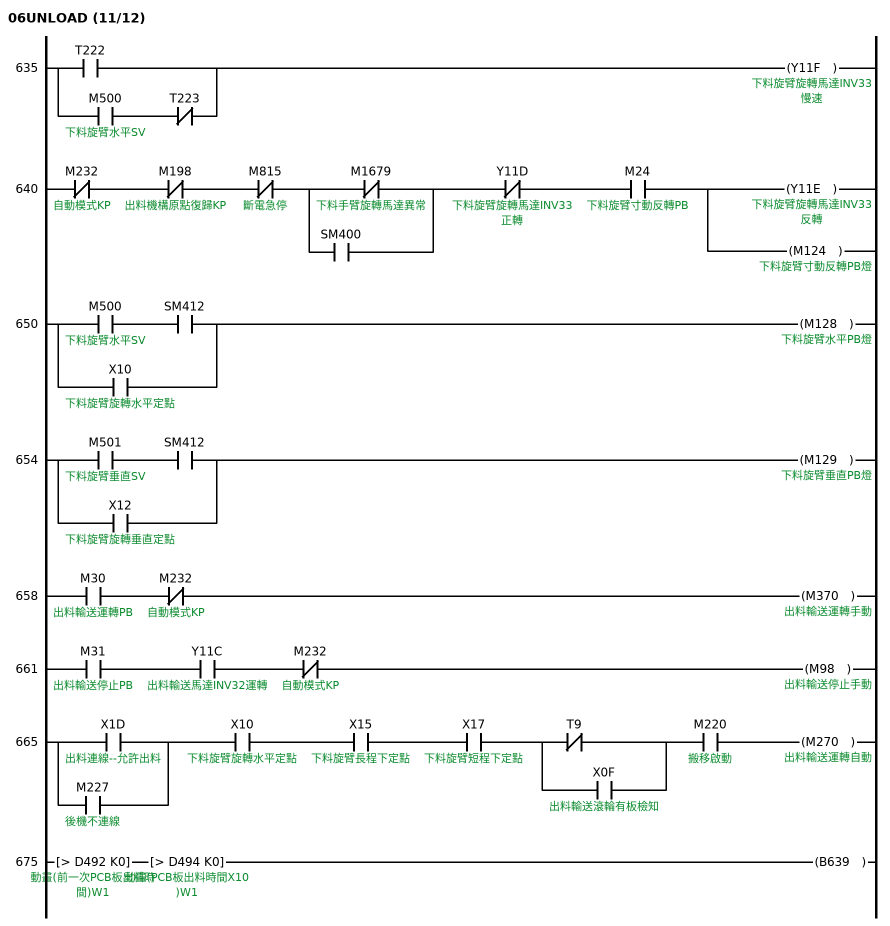
635   LD      T222
      LD      M500  ; 下料旋臂水平SV
      ANI     T223
      ORB
      OUT     Y11F  ; 下料旋臂旋轉馬達INV33慢速
640   LDI     M232  ; 自動模式KP
      ANI     M198  ; 出料機構原點復歸KP
      ANI     M815  ; 斷電急停
      LDI     M1679  ; 下料手臂旋轉馬達異常
      OR      SM400
      ANB
      ANI     Y11D  ; 下料旋臂旋轉馬達INV33正轉
      AND     M24  ; 下料旋臂寸動反轉PB
      OUT     Y11E  ; 下料旋臂旋轉馬達INV33反轉
      OUT     M124  ; 下料旋臂寸動反轉PB燈
650   LD      M500  ; 下料旋臂水平SV
      AND     SM412
      OR      X10  ; 下料旋臂旋轉水平定點
      OUT     M128  ; 下料旋臂水平PB燈
654   LD      M501  ; 下料旋臂垂直SV
      AND     SM412
      OR      X12  ; 下料旋臂旋轉垂直定點
      OUT     M129  ; 下料旋臂垂直PB燈
658   LD      M30  ; 出料輸送運轉PB
      ANI     M232  ; 自動模式KP
      OUT     M370  ; 出料輸送運轉手動
661   LD      M31  ; 出料輸送停止PB
      AND     Y11C  ; 出料輸送馬達INV32運轉
      ANI     M232  ; 自動模式KP
      OUT     M98  ; 出料輸送停止手動
665   LD      X1D  ; 出料連線--允許出料
      OR      M227  ; 後機不連線
      AND     X10  ; 下料旋臂旋轉水平定點
      AND     X15  ; 下料旋臂長程下定點
      AND     X17  ; 下料旋臂短程下定點
      LDI     T9
      OR      X0F  ; 出料輸送滾輪有板檢知
      ANB
      AND     M220  ; 搬移啟動
      OUT     M270  ; 出料輸送運轉自動
675   LD>     D492 K0  ; 動畫(前一次PCB板出料時間)W1
      AND>    D494 K0  ; 動畫(PCB板出料時間X10)W1
      OUT     B639
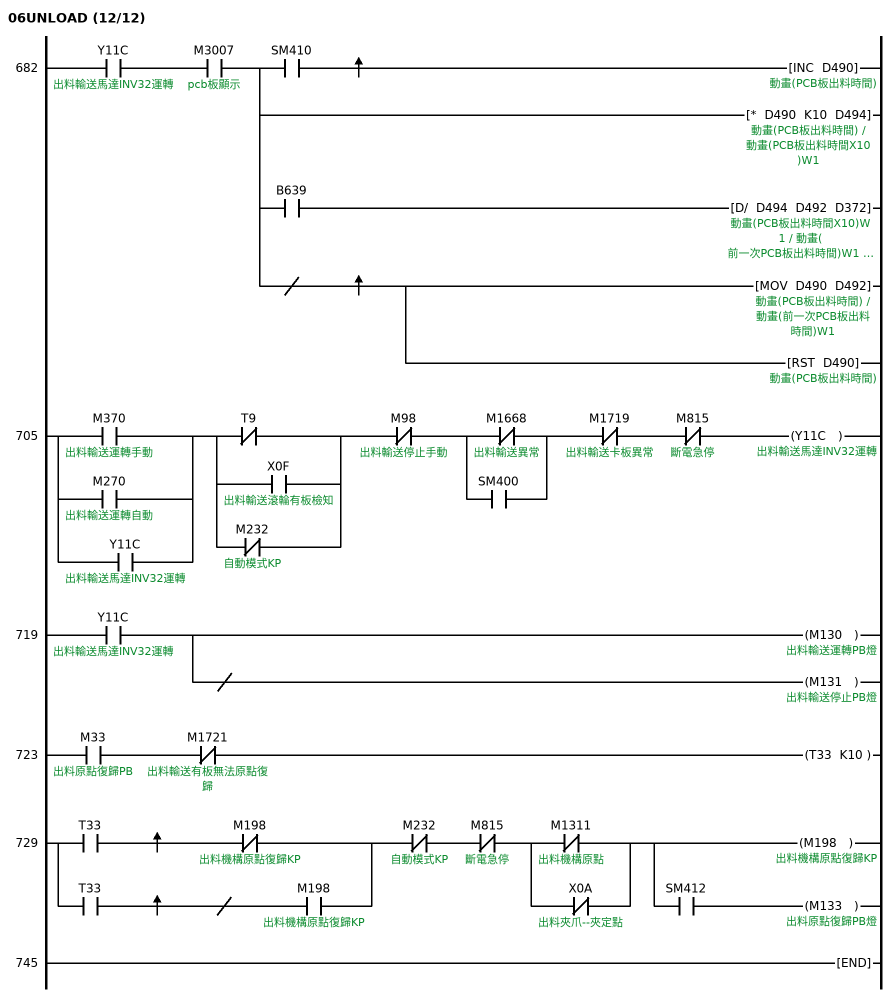
682   LD      Y11C  ; 出料輸送馬達INV32運轉
      AND     M3007  ; pcb板顯示
      MPS
      AND     SM410
      MEP
      INC     D490  ; 動畫(PCB板出料時間)
      MPP
      *       D490 K10 D494
      MPS
      AND     B639
      D/      D494 D492 D372  ; 動畫(PCB板出料現在位置)W1
      MPP
      INV
      MEP
      MOV     D490 D492
      RST     D490  ; 動畫(PCB板出料時間)
705   LD      M370  ; 出料輸送運轉手動
      OR      M270  ; 出料輸送運轉自動
      OR      Y11C  ; 出料輸送馬達INV32運轉
      LDI     T9
      OR      X0F  ; 出料輸送滾輪有板檢知
      ORI     M232  ; 自動模式KP
      ANB
      ANI     M98  ; 出料輸送停止手動
      LDI     M1668  ; 出料輸送異常
      OR      SM400
      ANB
      ANI     M1719  ; 出料輸送卡板異常
      ANI     M815  ; 斷電急停
      OUT     Y11C  ; 出料輸送馬達INV32運轉
719   LD      Y11C  ; 出料輸送馬達INV32運轉
      OUT     M130  ; 出料輸送運轉PB燈
      INV
      OUT     M131  ; 出料輸送停止PB燈
723   LD      M33  ; 出料原點復歸PB
      ANI     M1721  ; 出料輸送有板無法原點復歸
      OUT     T33 K10
729   LD      T33
      MEP
      ANI     M198  ; 出料機構原點復歸KP
      LD      T33
      MEP
      INV
      AND     M198  ; 出料機構原點復歸KP
      ORB
      ANI     M232  ; 自動模式KP
      ANI     M815  ; 斷電急停
      LDI     M1311  ; 出料機構原點
      ORI     X0A  ; 出料夾爪--夾定點
      ANB
      OUT     M198  ; 出料機構原點復歸KP
      AND     SM412
      OUT     M133  ; 出料原點復歸PB燈
745   END
END_PROGRAM

PROGRAM 07UNMOVE
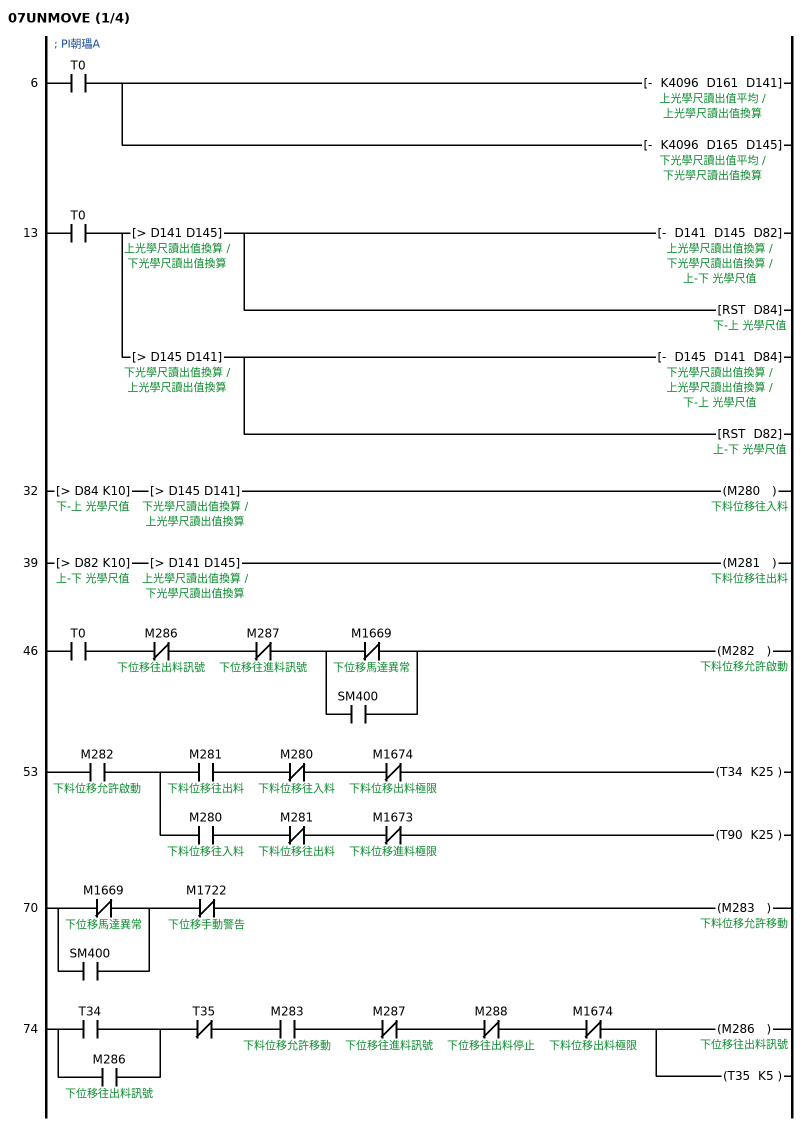
; PI朝瓃Α
6     LD      T0
      -       K4096 D161 D141  ; 上光學尺讀出值平均 / 上光學尺讀出值換算
      -       K4096 D165 D145  ; 下光學尺讀出值平均 / 下光學尺讀出值換算
13    LD      T0
      MPS
      AND>    D141 D145  ; 上光學尺讀出值換算 / 下光學尺讀出值換算
      -       D141 D145 D82  ; 上-下 光學尺值
      RST     D84  ; 下-上 光學尺值
      MPP
      AND>    D145 D141  ; 下光學尺讀出值換算 / 上光學尺讀出值換算
      -       D145 D141 D84
      RST     D82  ; 上-下 光學尺值
32    LD>     D84 K10  ; 下-上 光學尺值
      AND>    D145 D141  ; 下光學尺讀出值換算 / 上光學尺讀出值換算
      OUT     M280  ; 下料位移往入料
39    LD>     D82 K10  ; 上-下 光學尺值
      AND>    D141 D145  ; 上光學尺讀出值換算 / 下光學尺讀出值換算
      OUT     M281  ; 下料位移往出料
46    LD      T0
      ANI     M286  ; 下位移往出料訊號
      ANI     M287  ; 下位移往進料訊號
      LDI     M1669  ; 下位移馬達異常
      OR      SM400
      ANB
      OUT     M282  ; 下料位移允許啟動
53    LD      M282  ; 下料位移允許啟動
      MPS
      AND     M281  ; 下料位移往出料
      ANI     M280  ; 下料位移往入料
      ANI     M1674  ; 下料位移出料極限
      OUT     T34 K25
      MPP
      AND     M280  ; 下料位移往入料
      ANI     M281  ; 下料位移往出料
      ANI     M1673  ; 下料位移進料極限
      OUT     T90 K25
70    LDI     M1669  ; 下位移馬達異常
      OR      SM400
      ANI     M1722  ; 下位移手動警告
      OUT     M283  ; 下料位移允許移動
74    LD      T34
      OR      M286  ; 下位移往出料訊號
      ANI     T35
      AND     M283  ; 下料位移允許移動
      ANI     M287  ; 下位移往進料訊號
      ANI     M288  ; 下位移往出料停止
      ANI     M1674  ; 下料位移出料極限
      OUT     M286  ; 下位移往出料訊號
      OUT     T35 K5
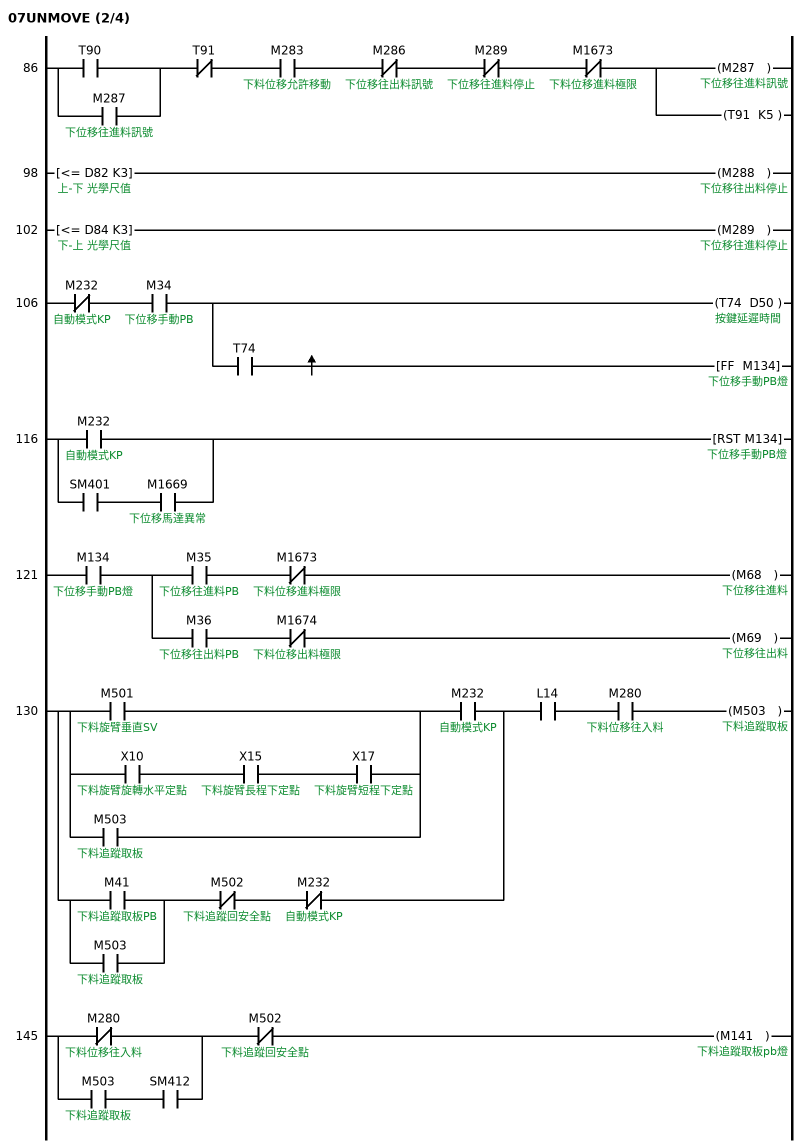
86    LD      T90
      OR      M287  ; 下位移往進料訊號
      ANI     T91
      AND     M283  ; 下料位移允許移動
      ANI     M286  ; 下位移往出料訊號
      ANI     M289  ; 下位移往進料停止
      ANI     M1673  ; 下料位移進料極限
      OUT     M287  ; 下位移往進料訊號
      OUT     T91 K5
98    LD<=    D82 K3  ; 上-下 光學尺值
      OUT     M288  ; 下位移往出料停止
102   LD<=    D84 K3  ; 下-上 光學尺值
      OUT     M289  ; 下位移往進料停止
106   LDI     M232  ; 自動模式KP
      AND     M34  ; 下位移手動PB
      OUT     T74 D50  ; 按鍵延遲時間
      AND     T74
      MEP
      FF      M134  ; 下位移手動PB燈
116   LD      M232  ; 自動模式KP
      LD      SM401
      AND     M1669  ; 下位移馬達異常
      ORB
      RST     M134  ; 下位移手動PB燈
121   LD      M134  ; 下位移手動PB燈
      MPS
      AND     M35  ; 下位移往進料PB
      ANI     M1673  ; 下料位移進料極限
      OUT     M68  ; 下位移往進料
      MPP
      AND     M36  ; 下位移往出料PB
      ANI     M1674  ; 下料位移出料極限
      OUT     M69  ; 下位移往出料
130   LD      M501  ; 下料旋臂垂直SV
      LD      X10  ; 下料旋臂旋轉水平定點
      AND     X15  ; 下料旋臂長程下定點
      AND     X17  ; 下料旋臂短程下定點
      ORB
      OR      M503  ; 下料追蹤取板
      AND     M232  ; 自動模式KP
      LD      M41  ; 下料追蹤取板PB
      OR      M503  ; 下料追蹤取板
      ANI     M502  ; 下料追蹤回安全點
      ANI     M232  ; 自動模式KP
      ORB
      AND     L14
      AND     M280  ; 下料位移往入料
      OUT     M503  ; 下料追蹤取板
145   LDI     M280  ; 下料位移往入料
      LD      M503  ; 下料追蹤取板
      AND     SM412
      ORB
      ANI     M502  ; 下料追蹤回安全點
      OUT     M141  ; 下料追蹤取板pb燈
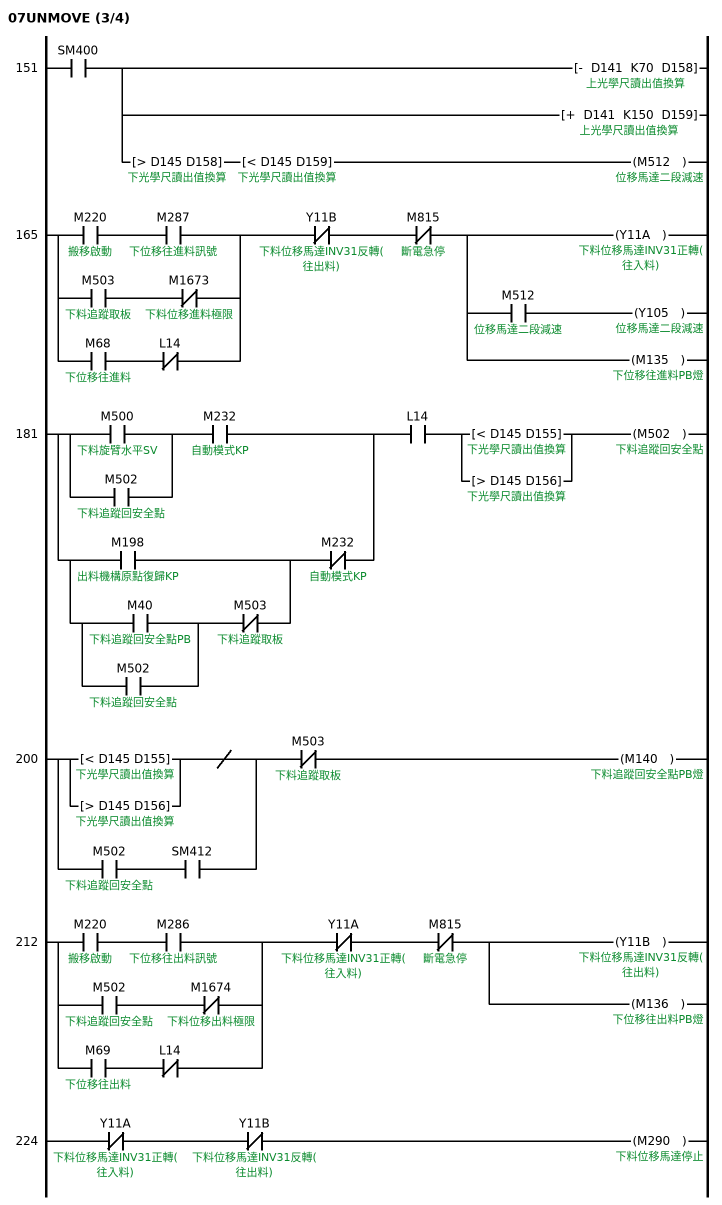
151   LD      SM400
      -       D141 K70 D158
      +       D141 K150 D159
      AND>    D145 D158  ; 下光學尺讀出值換算
      AND<    D145 D159  ; 下光學尺讀出值換算
      OUT     M512  ; 位移馬達二段減速
165   LD      M220  ; 搬移啟動
      AND     M287  ; 下位移往進料訊號
      LD      M503  ; 下料追蹤取板
      ANI     M1673  ; 下料位移進料極限
      ORB
      LD      M68  ; 下位移往進料
      ANI     L14
      ORB
      ANI     Y11B  ; 下料位移馬達INV31反轉(往出料)
      ANI     M815  ; 斷電急停
      OUT     Y11A  ; 下料位移馬達INV31正轉(往入料)
      MPS
      AND     M512  ; 位移馬達二段減速
      OUT     Y105  ; 位移馬達二段減速
      MPP
      OUT     M135  ; 下位移往進料PB燈
181   LD      M500  ; 下料旋臂水平SV
      OR      M502  ; 下料追蹤回安全點
      AND     M232  ; 自動模式KP
      LD      M198  ; 出料機構原點復歸KP
      LD      M40  ; 下料追蹤回安全點PB
      OR      M502  ; 下料追蹤回安全點
      ANI     M503  ; 下料追蹤取板
      ORB
      ANI     M232  ; 自動模式KP
      ORB
      AND     L14
      LD<     D145 D155  ; 下光學尺讀出值換算
      OR>     D145 D156  ; 下光學尺讀出值換算
      ANB
      OUT     M502  ; 下料追蹤回安全點
200   LD<     D145 D155  ; 下光學尺讀出值換算
      OR>     D145 D156  ; 下光學尺讀出值換算
      INV
      LD      M502  ; 下料追蹤回安全點
      AND     SM412
      ORB
      ANI     M503  ; 下料追蹤取板
      OUT     M140  ; 下料追蹤回安全點PB燈
212   LD      M220  ; 搬移啟動
      AND     M286  ; 下位移往出料訊號
      LD      M502  ; 下料追蹤回安全點
      ANI     M1674  ; 下料位移出料極限
      ORB
      LD      M69  ; 下位移往出料
      ANI     L14
      ORB
      ANI     Y11A  ; 下料位移馬達INV31正轉(往入料)
      ANI     M815  ; 斷電急停
      OUT     Y11B  ; 下料位移馬達INV31反轉(往出料)
      OUT     M136  ; 下位移往出料PB燈
224   LDI     Y11A  ; 下料位移馬達INV31正轉(往入料)
      ANI     Y11B  ; 下料位移馬達INV31反轉(往出料)
      OUT     M290  ; 下料位移馬達停止
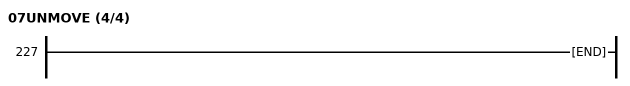
227   END
END_PROGRAM

PROGRAM 08HEATER
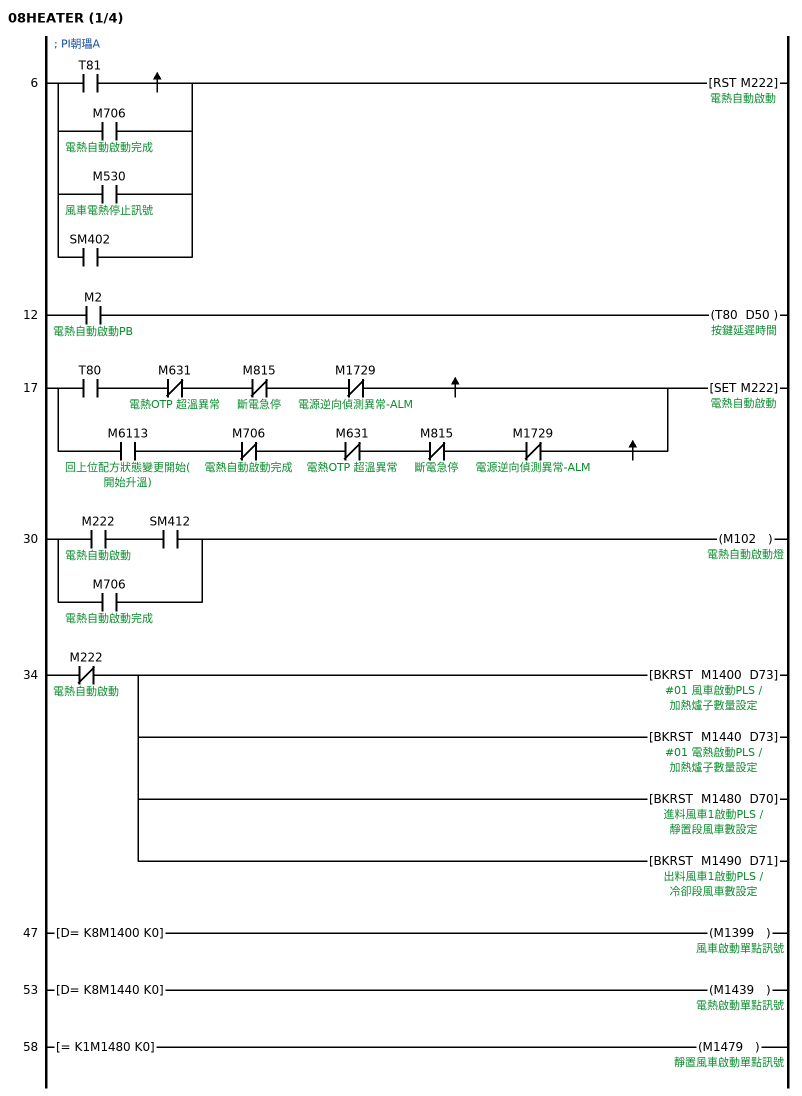
; PI朝瓃Α
6     LD      T81
      MEP
      OR      M706  ; 電熱自動啟動完成
      OR      M530  ; 風車電熱停止訊號
      OR      SM402
      RST     M222  ; 電熱自動啟動
12    LD      M2  ; 電熱自動啟動PB
      OUT     T80 D50  ; 按鍵延遲時間
17    LD      T80
      ANI     M631  ; 電熱OTP 超溫異常
      ANI     M815  ; 斷電急停
      ANI     M1729  ; 電源逆向偵測異常-ALM
      MEP
      LD      M6113  ; 回上位配方狀態變更開始(開始升溫)
      ANI     M706  ; 電熱自動啟動完成
      ANI     M631  ; 電熱OTP 超溫異常
      ANI     M815  ; 斷電急停
      ANI     M1729  ; 電源逆向偵測異常-ALM
      MEP
      ORB
      SET     M222  ; 電熱自動啟動
30    LD      M222  ; 電熱自動啟動
      AND     SM412
      OR      M706  ; 電熱自動啟動完成
      OUT     M102  ; 電熱自動啟動燈
34    LDI     M222  ; 電熱自動啟動
      BKRST   M1400 D73  ; #01 風車啟動PLS / 加熱爐子數量設定
      BKRST   M1440 D73  ; #01 電熱啟動PLS
      BKRST   M1480 D70  ; 進料風車1啟動PLS / 靜置段風車數設定
      BKRST   M1490 D71  ; 出料風車1啟動PLS / 冷卻段風車數設定
47    LDD=    K8M1400 K0  ; #01 風車啟動PLS
      OUT     M1399  ; 風車啟動單點訊號
53    LDD=    K8M1440 K0  ; #01 電熱啟動PLS
      OUT     M1439  ; 電熱啟動單點訊號
58    LD=     K1M1480 K0  ; 進料風車1啟動PLS
      OUT     M1479  ; 靜置風車啟動單點訊號
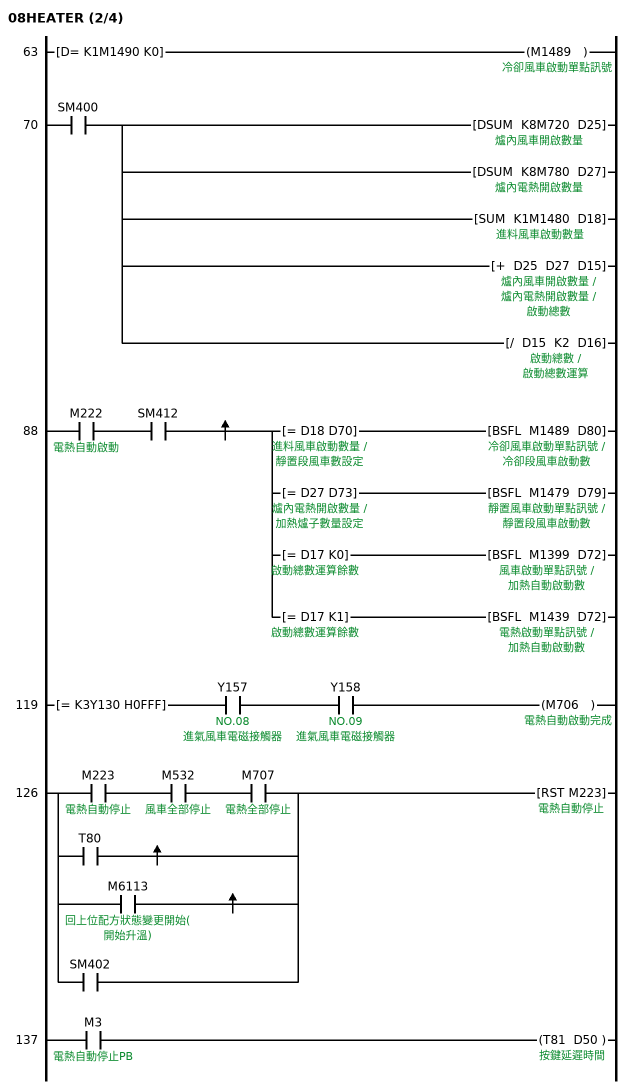
63    LDD=    K1M1490 K0  ; 出料風車1啟動PLS
      OUT     M1489  ; 冷卻風車啟動單點訊號
70    LD      SM400
      DSUM    K8M720 D25  ; #01 風車訊號 / 爐內風車開啟數量
      DSUM    K8M780 D27  ; #01 電熱訊號 / 爐內電熱開啟數量
      SUM     K1M1480 D18  ; 進料風車啟動數量
      +       D25 D27 D15  ; 啟動總數
      /       D15 K2 D16  ; 啟動總數運算
88    LD      M222  ; 電熱自動啟動
      AND     SM412
      MEP
      MPS
      AND=    D18 D70  ; 進料風車啟動數量 / 靜置段風車數設定
      BSFL    M1489 D80  ; 冷卻段風車啟動數
      MRD
      AND=    D27 D73  ; 爐內電熱開啟數量 / 加熱爐子數量設定
      BSFL    M1479 D79  ; 靜置段風車啟動數
      MRD
      AND=    D17 K0  ; 啟動總數運算餘數
      BSFL    M1399 D72  ; 加熱自動啟動數
      MPP
      AND=    D17 K1  ; 啟動總數運算餘數
      BSFL    M1439 D72
119   LD=     K3Y130 H0FFF  ; NO.01   加熱器電磁接觸器
      AND     Y157  ; NO.08   進氣風車電磁接觸器
      AND     Y158  ; NO.09   進氣風車電磁接觸器
      OUT     M706  ; 電熱自動啟動完成
126   LD      M223  ; 電熱自動停止
      AND     M532  ; 風車全部停止
      AND     M707  ; 電熱全部停止
      LD      T80
      MEP
      ORB
      LD      M6113  ; 回上位配方狀態變更開始(開始升溫)
      MEP
      ORB
      OR      SM402
      RST     M223  ; 電熱自動停止
137   LD      M3  ; 電熱自動停止PB
      OUT     T81 D50  ; 按鍵延遲時間
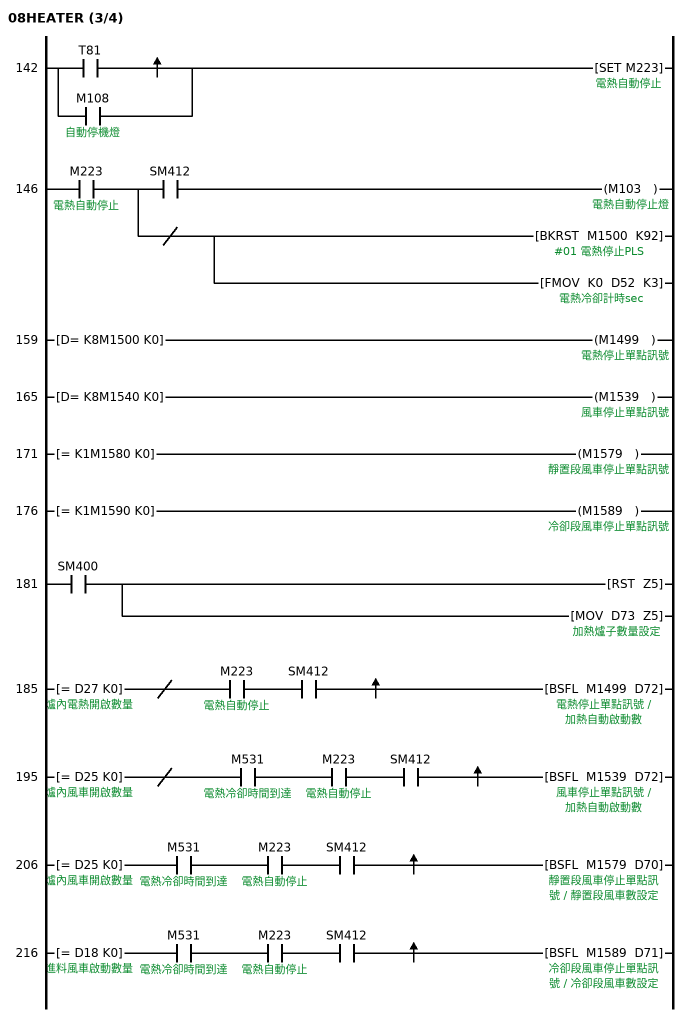
142   LD      T81
      MEP
      OR      M108  ; 自動停機燈
      SET     M223  ; 電熱自動停止
146   LD      M223  ; 電熱自動停止
      MPS
      AND     SM412
      OUT     M103  ; 電熱自動停止燈
      MPP
      INV
      BKRST   M1500 K92  ; #01 電熱停止PLS
      FMOV    K0 D52 K3  ; 電熱冷卻計時sec
159   LDD=    K8M1500 K0  ; #01 電熱停止PLS
      OUT     M1499  ; 電熱停止單點訊號
165   LDD=    K8M1540 K0  ; #01 風車停止PLS
      OUT     M1539  ; 風車停止單點訊號
171   LD=     K1M1580 K0  ; 進料風車1停止PLS
      OUT     M1579  ; 靜置段風車停止單點訊號
176   LD=     K1M1590 K0  ; 出料風車1停止PLS
      OUT     M1589  ; 冷卻段風車停止單點訊號
181   LD      SM400
      RST     Z5
      MOV     D73 Z5
185   LD=     D27 K0  ; 爐內電熱開啟數量
      INV
      AND     M223  ; 電熱自動停止
      AND     SM412
      MEP
      BSFL    M1499 D72
195   LD=     D25 K0  ; 爐內風車開啟數量
      INV
      AND     M531  ; 電熱冷卻時間到達
      AND     M223  ; 電熱自動停止
      AND     SM412
      MEP
      BSFL    M1539 D72
206   LD=     D25 K0  ; 爐內風車開啟數量
      AND     M531  ; 電熱冷卻時間到達
      AND     M223  ; 電熱自動停止
      AND     SM412
      MEP
      BSFL    M1579 D70
216   LD=     D18 K0  ; 進料風車啟動數量
      AND     M531  ; 電熱冷卻時間到達
      AND     M223  ; 電熱自動停止
      AND     SM412
      MEP
      BSFL    M1589 D71
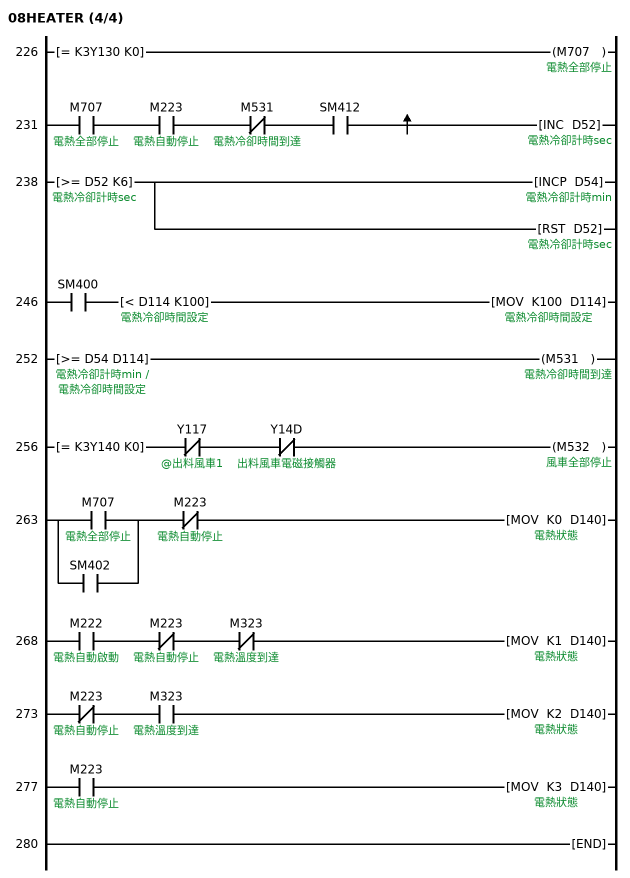
226   LD=     K3Y130 K0  ; NO.01   加熱器電磁接觸器
      OUT     M707  ; 電熱全部停止
231   LD      M707  ; 電熱全部停止
      AND     M223  ; 電熱自動停止
      ANI     M531  ; 電熱冷卻時間到達
      AND     SM412
      MEP
      INC     D52
238   LD>=    D52 K6  ; 電熱冷卻計時sec
      INCP    D54  ; 電熱冷卻計時min
      RST     D52  ; 電熱冷卻計時sec
246   LD      SM400
      AND<    D114 K100  ; 電熱冷卻時間設定
      MOV     K100 D114
252   LD>=    D54 D114  ; 電熱冷卻計時min / 電熱冷卻時間設定
      OUT     M531  ; 電熱冷卻時間到達
256   LD=     K3Y140 K0  ; NO.01   風車電磁接觸器
      ANI     Y117  ; @出料風車1
      ANI     Y14D  ; 出料風車電磁接觸器
      OUT     M532  ; 風車全部停止
263   LD      M707  ; 電熱全部停止
      OR      SM402
      ANI     M223  ; 電熱自動停止
      MOV     K0 D140  ; 電熱狀態
268   LD      M222  ; 電熱自動啟動
      ANI     M223  ; 電熱自動停止
      ANI     M323  ; 電熱溫度到達
      MOV     K1 D140
273   LDI     M223  ; 電熱自動停止
      AND     M323  ; 電熱溫度到達
      MOV     K2 D140
277   LD      M223  ; 電熱自動停止
      MOV     K3 D140
280   END
END_PROGRAM

PROGRAM 09BLOWER
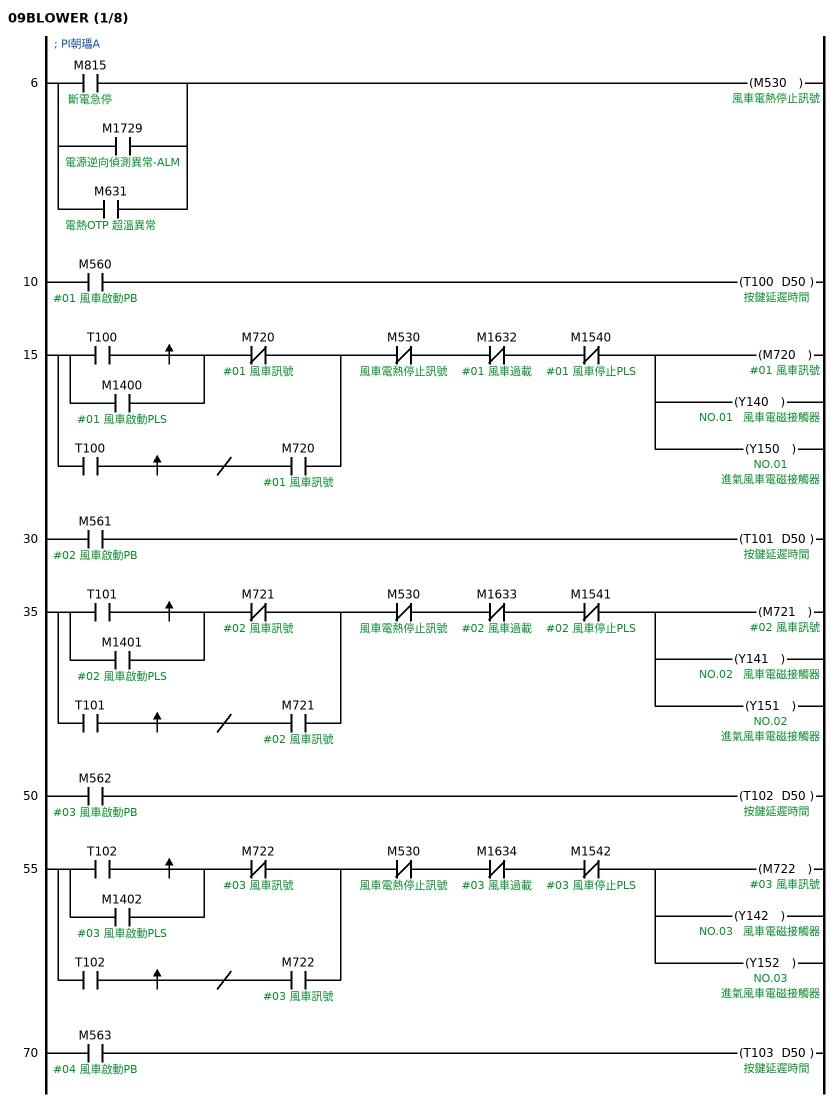
; PI朝瓃Α
6     LD      M815  ; 斷電急停
      OR      M1729  ; 電源逆向偵測異常-ALM
      OR      M631  ; 電熱OTP 超溫異常
      OUT     M530  ; 風車電熱停止訊號
10    LD      M560  ; #01 風車啟動PB
      OUT     T100 D50  ; 按鍵延遲時間
15    LD      T100
      MEP
      OR      M1400  ; #01 風車啟動PLS
      ANI     M720  ; #01 風車訊號
      LD      T100
      MEP
      INV
      AND     M720  ; #01 風車訊號
      ORB
      ANI     M530  ; 風車電熱停止訊號
      ANI     M1632  ; #01 風車過載
      ANI     M1540  ; #01 風車停止PLS
      OUT     M720  ; #01 風車訊號
      OUT     Y140  ; NO.01   風車電磁接觸器
      OUT     Y150  ; NO.01   進氣風車電磁接觸器
30    LD      M561  ; #02 風車啟動PB
      OUT     T101 D50  ; 按鍵延遲時間
35    LD      T101
      MEP
      OR      M1401  ; #02 風車啟動PLS
      ANI     M721  ; #02 風車訊號
      LD      T101
      MEP
      INV
      AND     M721  ; #02 風車訊號
      ORB
      ANI     M530  ; 風車電熱停止訊號
      ANI     M1633  ; #02 風車過載
      ANI     M1541  ; #02 風車停止PLS
      OUT     M721  ; #02 風車訊號
      OUT     Y141  ; NO.02   風車電磁接觸器
      OUT     Y151  ; NO.02   進氣風車電磁接觸器
50    LD      M562  ; #03 風車啟動PB
      OUT     T102 D50  ; 按鍵延遲時間
55    LD      T102
      MEP
      OR      M1402  ; #03 風車啟動PLS
      ANI     M722  ; #03 風車訊號
      LD      T102
      MEP
      INV
      AND     M722  ; #03 風車訊號
      ORB
      ANI     M530  ; 風車電熱停止訊號
      ANI     M1634  ; #03 風車過載
      ANI     M1542  ; #03 風車停止PLS
      OUT     M722  ; #03 風車訊號
      OUT     Y142  ; NO.03   風車電磁接觸器
      OUT     Y152  ; NO.03   進氣風車電磁接觸器
70    LD      M563  ; #04 風車啟動PB
      OUT     T103 D50  ; 按鍵延遲時間
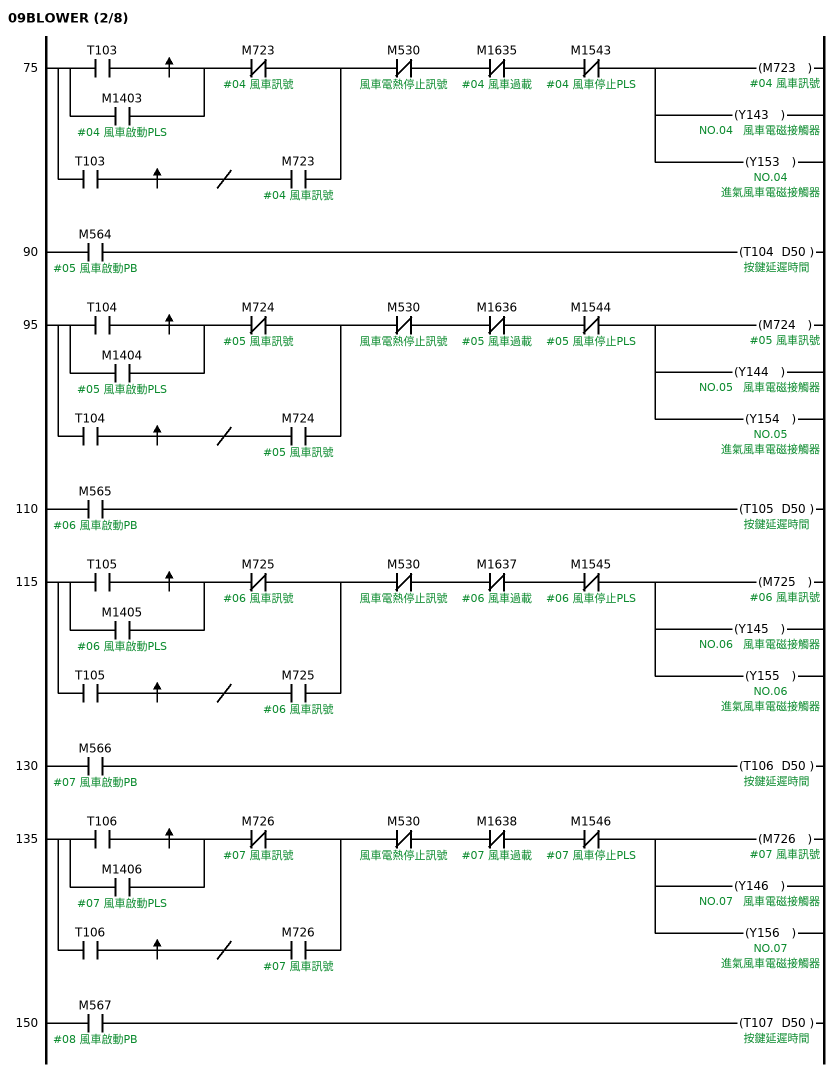
75    LD      T103
      MEP
      OR      M1403  ; #04 風車啟動PLS
      ANI     M723  ; #04 風車訊號
      LD      T103
      MEP
      INV
      AND     M723  ; #04 風車訊號
      ORB
      ANI     M530  ; 風車電熱停止訊號
      ANI     M1635  ; #04 風車過載
      ANI     M1543  ; #04 風車停止PLS
      OUT     M723  ; #04 風車訊號
      OUT     Y143  ; NO.04   風車電磁接觸器
      OUT     Y153  ; NO.04   進氣風車電磁接觸器
90    LD      M564  ; #05 風車啟動PB
      OUT     T104 D50  ; 按鍵延遲時間
95    LD      T104
      MEP
      OR      M1404  ; #05 風車啟動PLS
      ANI     M724  ; #05 風車訊號
      LD      T104
      MEP
      INV
      AND     M724  ; #05 風車訊號
      ORB
      ANI     M530  ; 風車電熱停止訊號
      ANI     M1636  ; #05 風車過載
      ANI     M1544  ; #05 風車停止PLS
      OUT     M724  ; #05 風車訊號
      OUT     Y144  ; NO.05   風車電磁接觸器
      OUT     Y154  ; NO.05   進氣風車電磁接觸器
110   LD      M565  ; #06 風車啟動PB
      OUT     T105 D50  ; 按鍵延遲時間
115   LD      T105
      MEP
      OR      M1405  ; #06 風車啟動PLS
      ANI     M725  ; #06 風車訊號
      LD      T105
      MEP
      INV
      AND     M725  ; #06 風車訊號
      ORB
      ANI     M530  ; 風車電熱停止訊號
      ANI     M1637  ; #06 風車過載
      ANI     M1545  ; #06 風車停止PLS
      OUT     M725  ; #06 風車訊號
      OUT     Y145  ; NO.06   風車電磁接觸器
      OUT     Y155  ; NO.06   進氣風車電磁接觸器
130   LD      M566  ; #07 風車啟動PB
      OUT     T106 D50  ; 按鍵延遲時間
135   LD      T106
      MEP
      OR      M1406  ; #07 風車啟動PLS
      ANI     M726  ; #07 風車訊號
      LD      T106
      MEP
      INV
      AND     M726  ; #07 風車訊號
      ORB
      ANI     M530  ; 風車電熱停止訊號
      ANI     M1638  ; #07 風車過載
      ANI     M1546  ; #07 風車停止PLS
      OUT     M726  ; #07 風車訊號
      OUT     Y146  ; NO.07   風車電磁接觸器
      OUT     Y156  ; NO.07   進氣風車電磁接觸器
150   LD      M567  ; #08 風車啟動PB
      OUT     T107 D50  ; 按鍵延遲時間
